// TIA Portal V20 export
DATA_BLOCK "HmiInterface"   // DB98
{ DB_Accessible_From_OPC_UA := 'FALSE' }
AUTHOR : ERsystem_FA2_DH. Kim
// stored: Access Published, DBAccessibleFromOPCUA false, DBAccessibleFromWebserver false, MemoryReserve 100, Namespace Unit1.Em5
   VAR
      em : "LAF_typeEmInterface";
      cm : Struct
         softCam : "Unit1.type_emRelations_em5_SoftCam";
         brakeTest : Struct
            cathodeMainPnP1AxisZ : "LER_typeBrakeTestEmInterface";
            cathodeMainPnP2AxisZ : "LER_typeBrakeTestEmInterface";
         END_STRUCT;
      END_STRUCT;
      mainPnP : Struct
         jobs { S7_SetPoint := 'True'} : "LAF_typeJobsInterface";
         sequence { S7_SetPoint := 'True'} : "LAF_typeSequenceInterface";
      END_STRUCT;
      alignTable : Struct
         jobs { S7_SetPoint := 'True'} : "LAF_typeJobsInterface";
         sequence { S7_SetPoint := 'True'} : "LAF_typeSequenceInterface";
      END_STRUCT;
      ngPnP : Struct
         jobs { S7_SetPoint := 'True'} : "LAF_typeJobsInterface";
         sequence { S7_SetPoint := 'True'} : "LAF_typeSequenceInterface";
      END_STRUCT;
      gaugeRnR : Struct
         jobs { S7_SetPoint := 'True'} : "LAF_typeJobsInterface";
         sequence { S7_SetPoint := 'True'} : "LAF_typeSequenceInterface";
      END_STRUCT;
      cathodeNgCount : "LER_typeAlarmCounterInterface";
      cmPnp1stCathodeDetect { S7_SetPoint := 'True'} : "LBC_typeDigitalSignalInterface";
      cmPnp2ndCathodeDetect { S7_SetPoint := 'True'} : "LBC_typeDigitalSignalInterface";
      cmCathodeAlignTableElectrodeDetect { S7_SetPoint := 'True'} : "LBC_typeDigitalSignalInterface";
      cmCathodeNgPnpElectrodeDetect { S7_SetPoint := 'True'} : "LBC_typeDigitalSignalInterface";
      cmCathodeNgBoxFullSensorDetect { S7_SetPoint := 'True'} : "LBC_typeDigitalSignalInterface";
      cmCathodeNgBoxDetect { S7_SetPoint := 'True'} : "LBC_typeDigitalSignalInterface";
   END_VAR
   VAR RETAIN
      cmCathodeMainPnP1AxisX : "LBC_typeAxis64PosInterface";
      cmCathodeMainPnP2AxisX : "LBC_typeAxis64PosInterface";
      cmCathodeMainPnP1AxisY : "LBC_typeAxis64PosInterface";
      cmCathodeMainPnP1AxisZ : "LBC_typeAxis64PosInterface";
      cmCathodeMainPnP2AxisZ : "LBC_typeAxis64PosInterface";
      cmCathodeAlignTableAxisX : "LBC_typeAxis64PosInterface";
      cmCathodeAlignTableAxisY1 : "LBC_typeAxis64PosInterface";
      cmCathodeAlignTableAxisY2 : "LBC_typeAxis64PosInterface";
   END_VAR
   VAR
      cmCathodeMainPnP1RotaryCwCcw : "LBC_typeTwoWayActuatorInterface";
      cmCathodeMainPnP1SuctionPlateVacuum : "LBC_typeTwoWayActuatorInterface";
      cmCathodeMainPnP2SuctionPlateVacuum : "LBC_typeTwoWayActuatorInterface";
      cmCathodeAlignTableSuctionPlateVacuum : "LBC_typeTwoWayActuatorInterface";
      cmCathodeGlassCleaning : "LBC_typeTwoWayActuatorInterface";
      cmCathodeNgPnpUpDown : "LBC_typeTwoWayActuatorInterface";
      cmCathodeNgPnp1stFwdBwd : "LBC_typeTwoWayActuatorInterface";
      cmCathodeNgPnp2ndFwdBwd { S7_SetPoint := 'True'} : "LBC_typeTwoWayActuatorInterface";
      cmCathodeMaintenanceMovingFixFrontRearFwdBwd : "LBC_typeTwoWayActuatorInterface";
      cmCathodeNgBoxLiftUpDown { S7_SetPoint := 'True'} : "LBC_typeTwoWayActuatorInterface";
      cmCathodeNgBoxLockUpDown { S7_SetPoint := 'True'} : "LBC_typeTwoWayActuatorInterface";
      cmCathodeNgPnpVaccum : "LBC_typeTwoWayActuatorInterface";
      cmCathodeConveyorCoverFwdBwd { S7_SetPoint := 'True'} : "LBC_typeTwoWayActuatorInterface";
      cmCathodeConveyorPickUpBlower { S7_SetPoint := 'True'} : "LBC_typeTwoWayActuatorInterface";
      cmAlignVisionControllerInterface : "LER_typeVisionInterface";
      AlignVisionHistory : "LER_typeVisionHistory";
      AlignVisionConversion : "LER_typeVisionAlignResultData";
      AlignCalibration : "LER_typeAlignCalibrationInterface";
      AlignMoveCalibration : "LER_typeAlignMoveCalibrationInterface";
      AlignThetaCalibration { S7_SetPoint := 'True'} : "LER_typeAlignThetaCalibrationInterface";
      AlignSyncMove : "LER_typeAlignSyncMoveInterface";
   END_VAR
   VAR RETAIN
      GaugeRnR1Align : "LER_typeCount";
   END_VAR
   VAR
      GaugeRnR1Stack { S7_SetPoint := 'True'} : "LER_typeCount";
      GaugeRnR3Align { S7_SetPoint := 'True'} : "LER_typeCount";
      intCondition : Struct
         Axis_07 { S7_SetPoint := 'True'} : "LER.typeAxisIntlockAll";   // CathodeMainPnP1AxisX
         Axis_08 { S7_SetPoint := 'True'} : "LER.typeAxisIntlockAll";   // CathodeMainPnP2AxisX
         Axis_09 { S7_SetPoint := 'True'} : "LER.typeAxisIntlockAll";   // CathodeMainPnP1AxisY
         Axis_10 { S7_SetPoint := 'True'} : "LER.typeAxisIntlockAll";   // CathodeMainPnP1AxisZ
         Axis_13 { S7_SetPoint := 'True'} : "LER.typeAxisIntlockAll";   // CathodeMainPnP2AxisZ
         Axis_18 { S7_SetPoint := 'True'} : "LER.typeAxisIntlockAll";   // CathodeAlignTableAxisX
         Axis_19 { S7_SetPoint := 'True'} : "LER.typeAxisIntlockAll";   // CathodeAlignTableAxisY1
         Axis_20 { S7_SetPoint := 'True'} : "LER.typeAxisIntlockAll";   // CathodeAlignTableAxisY2
         Actuator_23 : "LER.typeAxisActuatorCondition";   // CathodeMaintenanceMovingFixFrontFwdBwd
         Actuator_24 : "LER.typeAxisActuatorCondition";   // SP
         Actuator_25 : "LER.typeAxisActuatorCondition";   // CathodeNgBoxLockUpDown
         Actuator_26 : "LER.typeAxisActuatorCondition";   // CathodeNgBoxLiftUpDown
         Actuator_27 : "LER.typeAxisActuatorCondition";   // CathodeNgPnp2ndFwdBwd
         Actuator_28 : "LER.typeAxisActuatorCondition";   // SP
         Actuator_29 : "LER.typeAxisActuatorCondition";   // CathodeNgPnpUpDown
         Actuator_30 : "LER.typeAxisActuatorCondition";   // CathodeGlassCleaning
         Actuator_31 : "LER.typeAxisActuatorCondition";   // CathodeMainPnP1RotaryCwCcw
         Actuator_32 : "LER.typeAxisActuatorCondition";   // CathodeNgPnp1stFwdBwd
      END_STRUCT;
   END_VAR
BEGIN
   em.interlinkMode.link := FALSE;
   em.interlinkMode.unlink := FALSE;
   em.interlinkMode.isLinked := TRUE;
   em.commands.enable := FALSE;
   em.commands.acknowledge := FALSE;
   em.commands.disableAlarms := FALSE;
   em.commands.activateSimulation := FALSE;
   em.commands.home := FALSE;
   em.commands.moveToInitialPosition := FALSE;
   em.commands.directModeControl := 16#0000_0001;
   em.commands.directStateControl := 16#0000_0004;
   em.status.enabled := TRUE;
   em.status.acknowledgeActive := FALSE;
   em.status.alarmsDisabled := FALSE;
   em.status.simulationActive := TRUE;
   em.status.safetyReleased := TRUE;
   em.status.initialized := TRUE;
   em.status.homed := FALSE;
   em.status.safeState := FALSE;
   em.status.stateComplete := FALSE;
   em.alarms.error := FALSE;
   em.alarms.warning := TRUE;
   em.alarms.info := FALSE;
   em.alarms.home := FALSE;
   cm.softCam.cathodeMainPnP1AxisX.reelCutConveyerPos.inPos := FALSE;
   cm.softCam.cathodeMainPnP1AxisX.reelCutConveyerPos.isBefore := FALSE;
   cm.softCam.cathodeMainPnP1AxisX.reelCutConveyerPos.isAfter := TRUE;
   cm.softCam.cathodeMainPnP1AxisX.alignTablePos.inPos := TRUE;
   cm.softCam.cathodeMainPnP1AxisX.alignTablePos.isBefore := FALSE;
   cm.softCam.cathodeMainPnP1AxisX.alignTablePos.isAfter := FALSE;
   cm.softCam.cathodeMainPnP1AxisX.Pos2.inPos := FALSE;
   cm.softCam.cathodeMainPnP1AxisX.Pos2.isBefore := TRUE;
   cm.softCam.cathodeMainPnP1AxisX.Pos2.isAfter := FALSE;
   cm.softCam.cathodeMainPnP1AxisX.Pos3.inPos := FALSE;
   cm.softCam.cathodeMainPnP1AxisX.Pos3.isBefore := FALSE;
   cm.softCam.cathodeMainPnP1AxisX.Pos3.isAfter := TRUE;
   cm.softCam.cathodeMainPnP1AxisX.Pos4.inPos := FALSE;
   cm.softCam.cathodeMainPnP1AxisX.Pos4.isBefore := FALSE;
   cm.softCam.cathodeMainPnP1AxisX.Pos4.isAfter := TRUE;
   cm.softCam.cathodeMainPnP1AxisX.Pos5.inPos := FALSE;
   cm.softCam.cathodeMainPnP1AxisX.Pos5.isBefore := FALSE;
   cm.softCam.cathodeMainPnP1AxisX.Pos5.isAfter := TRUE;
   cm.softCam.cathodeMainPnP1AxisX.Pos6.inPos := FALSE;
   cm.softCam.cathodeMainPnP1AxisX.Pos6.isBefore := FALSE;
   cm.softCam.cathodeMainPnP1AxisX.Pos6.isAfter := TRUE;
   cm.softCam.cathodeMainPnP1AxisX.Pos7.inPos := FALSE;
   cm.softCam.cathodeMainPnP1AxisX.Pos7.isBefore := FALSE;
   cm.softCam.cathodeMainPnP1AxisX.Pos7.isAfter := TRUE;
   cm.softCam.cathodeMainPnP1AxisX.Pos8.inPos := FALSE;
   cm.softCam.cathodeMainPnP1AxisX.Pos8.isBefore := FALSE;
   cm.softCam.cathodeMainPnP1AxisX.Pos8.isAfter := TRUE;
   cm.softCam.cathodeMainPnP1AxisX.Pos9.inPos := FALSE;
   cm.softCam.cathodeMainPnP1AxisX.Pos9.isBefore := FALSE;
   cm.softCam.cathodeMainPnP1AxisX.Pos9.isAfter := TRUE;
   cm.softCam.cathodeMainPnP1AxisX.Pos10.inPos := FALSE;
   cm.softCam.cathodeMainPnP1AxisX.Pos10.isBefore := FALSE;
   cm.softCam.cathodeMainPnP1AxisX.Pos10.isAfter := TRUE;
   cm.softCam.cathodeMainPnP1AxisX.Pos11.inPos := FALSE;
   cm.softCam.cathodeMainPnP1AxisX.Pos11.isBefore := FALSE;
   cm.softCam.cathodeMainPnP1AxisX.Pos11.isAfter := TRUE;
   cm.softCam.cathodeMainPnP1AxisX.Pos12.inPos := FALSE;
   cm.softCam.cathodeMainPnP1AxisX.Pos12.isBefore := FALSE;
   cm.softCam.cathodeMainPnP1AxisX.Pos12.isAfter := TRUE;
   cm.softCam.cathodeMainPnP1AxisX.Pos13.inPos := FALSE;
   cm.softCam.cathodeMainPnP1AxisX.Pos13.isBefore := FALSE;
   cm.softCam.cathodeMainPnP1AxisX.Pos13.isAfter := TRUE;
   cm.softCam.cathodeMainPnP1AxisX.Pos14.inPos := FALSE;
   cm.softCam.cathodeMainPnP1AxisX.Pos14.isBefore := FALSE;
   cm.softCam.cathodeMainPnP1AxisX.Pos14.isAfter := TRUE;
   cm.softCam.cathodeMainPnP1AxisX.Pos15.inPos := FALSE;
   cm.softCam.cathodeMainPnP1AxisX.Pos15.isBefore := FALSE;
   cm.softCam.cathodeMainPnP1AxisX.Pos15.isAfter := TRUE;
   cm.softCam.cathodeMainPnP2AxisX.alignTablePos.inPos := FALSE;
   cm.softCam.cathodeMainPnP2AxisX.alignTablePos.isBefore := FALSE;
   cm.softCam.cathodeMainPnP2AxisX.alignTablePos.isAfter := TRUE;
   cm.softCam.cathodeMainPnP2AxisX.stackTablePos.inPos := TRUE;
   cm.softCam.cathodeMainPnP2AxisX.stackTablePos.isBefore := FALSE;
   cm.softCam.cathodeMainPnP2AxisX.stackTablePos.isAfter := FALSE;
   cm.softCam.cathodeMainPnP2AxisX.Pos2.inPos := FALSE;
   cm.softCam.cathodeMainPnP2AxisX.Pos2.isBefore := FALSE;
   cm.softCam.cathodeMainPnP2AxisX.Pos2.isAfter := TRUE;
   cm.softCam.cathodeMainPnP2AxisX.Pos3.inPos := FALSE;
   cm.softCam.cathodeMainPnP2AxisX.Pos3.isBefore := FALSE;
   cm.softCam.cathodeMainPnP2AxisX.Pos3.isAfter := TRUE;
   cm.softCam.cathodeMainPnP2AxisX.Pos4.inPos := FALSE;
   cm.softCam.cathodeMainPnP2AxisX.Pos4.isBefore := FALSE;
   cm.softCam.cathodeMainPnP2AxisX.Pos4.isAfter := TRUE;
   cm.softCam.cathodeMainPnP2AxisX.Pos5.inPos := FALSE;
   cm.softCam.cathodeMainPnP2AxisX.Pos5.isBefore := FALSE;
   cm.softCam.cathodeMainPnP2AxisX.Pos5.isAfter := TRUE;
   cm.softCam.cathodeMainPnP2AxisX.Pos6.inPos := FALSE;
   cm.softCam.cathodeMainPnP2AxisX.Pos6.isBefore := FALSE;
   cm.softCam.cathodeMainPnP2AxisX.Pos6.isAfter := TRUE;
   cm.softCam.cathodeMainPnP2AxisX.Pos7.inPos := FALSE;
   cm.softCam.cathodeMainPnP2AxisX.Pos7.isBefore := FALSE;
   cm.softCam.cathodeMainPnP2AxisX.Pos7.isAfter := TRUE;
   cm.softCam.cathodeMainPnP2AxisX.Pos8.inPos := FALSE;
   cm.softCam.cathodeMainPnP2AxisX.Pos8.isBefore := FALSE;
   cm.softCam.cathodeMainPnP2AxisX.Pos8.isAfter := TRUE;
   cm.softCam.cathodeMainPnP2AxisX.Pos9.inPos := FALSE;
   cm.softCam.cathodeMainPnP2AxisX.Pos9.isBefore := FALSE;
   cm.softCam.cathodeMainPnP2AxisX.Pos9.isAfter := TRUE;
   cm.softCam.cathodeMainPnP2AxisX.Pos10.inPos := FALSE;
   cm.softCam.cathodeMainPnP2AxisX.Pos10.isBefore := FALSE;
   cm.softCam.cathodeMainPnP2AxisX.Pos10.isAfter := TRUE;
   cm.softCam.cathodeMainPnP2AxisX.Pos11.inPos := FALSE;
   cm.softCam.cathodeMainPnP2AxisX.Pos11.isBefore := FALSE;
   cm.softCam.cathodeMainPnP2AxisX.Pos11.isAfter := TRUE;
   cm.softCam.cathodeMainPnP2AxisX.Pos12.inPos := FALSE;
   cm.softCam.cathodeMainPnP2AxisX.Pos12.isBefore := FALSE;
   cm.softCam.cathodeMainPnP2AxisX.Pos12.isAfter := TRUE;
   cm.softCam.cathodeMainPnP2AxisX.Pos13.inPos := FALSE;
   cm.softCam.cathodeMainPnP2AxisX.Pos13.isBefore := FALSE;
   cm.softCam.cathodeMainPnP2AxisX.Pos13.isAfter := TRUE;
   cm.softCam.cathodeMainPnP2AxisX.Pos14.inPos := FALSE;
   cm.softCam.cathodeMainPnP2AxisX.Pos14.isBefore := FALSE;
   cm.softCam.cathodeMainPnP2AxisX.Pos14.isAfter := TRUE;
   cm.softCam.cathodeMainPnP2AxisX.Pos15.inPos := FALSE;
   cm.softCam.cathodeMainPnP2AxisX.Pos15.isBefore := FALSE;
   cm.softCam.cathodeMainPnP2AxisX.Pos15.isAfter := TRUE;
   cm.softCam.cathodeMainPnP1AxisY.waitPos.inPos := TRUE;
   cm.softCam.cathodeMainPnP1AxisY.waitPos.isBefore := FALSE;
   cm.softCam.cathodeMainPnP1AxisY.waitPos.isAfter := FALSE;
   cm.softCam.cathodeMainPnP1AxisY.Pos1.inPos := TRUE;
   cm.softCam.cathodeMainPnP1AxisY.Pos1.isBefore := FALSE;
   cm.softCam.cathodeMainPnP1AxisY.Pos1.isAfter := FALSE;
   cm.softCam.cathodeMainPnP1AxisY.Pos2.inPos := TRUE;
   cm.softCam.cathodeMainPnP1AxisY.Pos2.isBefore := FALSE;
   cm.softCam.cathodeMainPnP1AxisY.Pos2.isAfter := FALSE;
   cm.softCam.cathodeMainPnP1AxisY.Pos3.inPos := TRUE;
   cm.softCam.cathodeMainPnP1AxisY.Pos3.isBefore := FALSE;
   cm.softCam.cathodeMainPnP1AxisY.Pos3.isAfter := FALSE;
   cm.softCam.cathodeMainPnP1AxisY.Pos4.inPos := TRUE;
   cm.softCam.cathodeMainPnP1AxisY.Pos4.isBefore := FALSE;
   cm.softCam.cathodeMainPnP1AxisY.Pos4.isAfter := FALSE;
   cm.softCam.cathodeMainPnP1AxisY.Pos5.inPos := TRUE;
   cm.softCam.cathodeMainPnP1AxisY.Pos5.isBefore := FALSE;
   cm.softCam.cathodeMainPnP1AxisY.Pos5.isAfter := FALSE;
   cm.softCam.cathodeMainPnP1AxisY.Pos6.inPos := TRUE;
   cm.softCam.cathodeMainPnP1AxisY.Pos6.isBefore := FALSE;
   cm.softCam.cathodeMainPnP1AxisY.Pos6.isAfter := FALSE;
   cm.softCam.cathodeMainPnP1AxisY.Pos7.inPos := TRUE;
   cm.softCam.cathodeMainPnP1AxisY.Pos7.isBefore := FALSE;
   cm.softCam.cathodeMainPnP1AxisY.Pos7.isAfter := FALSE;
   cm.softCam.cathodeMainPnP1AxisY.Pos8.inPos := TRUE;
   cm.softCam.cathodeMainPnP1AxisY.Pos8.isBefore := FALSE;
   cm.softCam.cathodeMainPnP1AxisY.Pos8.isAfter := FALSE;
   cm.softCam.cathodeMainPnP1AxisY.Pos9.inPos := TRUE;
   cm.softCam.cathodeMainPnP1AxisY.Pos9.isBefore := FALSE;
   cm.softCam.cathodeMainPnP1AxisY.Pos9.isAfter := FALSE;
   cm.softCam.cathodeMainPnP1AxisY.Pos10.inPos := TRUE;
   cm.softCam.cathodeMainPnP1AxisY.Pos10.isBefore := FALSE;
   cm.softCam.cathodeMainPnP1AxisY.Pos10.isAfter := FALSE;
   cm.softCam.cathodeMainPnP1AxisY.Pos11.inPos := TRUE;
   cm.softCam.cathodeMainPnP1AxisY.Pos11.isBefore := FALSE;
   cm.softCam.cathodeMainPnP1AxisY.Pos11.isAfter := FALSE;
   cm.softCam.cathodeMainPnP1AxisY.Pos12.inPos := TRUE;
   cm.softCam.cathodeMainPnP1AxisY.Pos12.isBefore := FALSE;
   cm.softCam.cathodeMainPnP1AxisY.Pos12.isAfter := FALSE;
   cm.softCam.cathodeMainPnP1AxisY.Pos13.inPos := TRUE;
   cm.softCam.cathodeMainPnP1AxisY.Pos13.isBefore := FALSE;
   cm.softCam.cathodeMainPnP1AxisY.Pos13.isAfter := FALSE;
   cm.softCam.cathodeMainPnP1AxisY.Pos14.inPos := TRUE;
   cm.softCam.cathodeMainPnP1AxisY.Pos14.isBefore := FALSE;
   cm.softCam.cathodeMainPnP1AxisY.Pos14.isAfter := FALSE;
   cm.softCam.cathodeMainPnP1AxisY.Pos15.inPos := TRUE;
   cm.softCam.cathodeMainPnP1AxisY.Pos15.isBefore := FALSE;
   cm.softCam.cathodeMainPnP1AxisY.Pos15.isAfter := FALSE;
   cm.softCam.cathodeMainPnP1AxisZ.upPos.inPos := FALSE;
   cm.softCam.cathodeMainPnP1AxisZ.upPos.isBefore := FALSE;
   cm.softCam.cathodeMainPnP1AxisZ.upPos.isAfter := TRUE;
   cm.softCam.cathodeMainPnP1AxisZ.reelCutConveyerDownPos.inPos := TRUE;
   cm.softCam.cathodeMainPnP1AxisZ.reelCutConveyerDownPos.isBefore := FALSE;
   cm.softCam.cathodeMainPnP1AxisZ.reelCutConveyerDownPos.isAfter := FALSE;
   cm.softCam.cathodeMainPnP1AxisZ.ailgnTableDownPos.inPos := TRUE;
   cm.softCam.cathodeMainPnP1AxisZ.ailgnTableDownPos.isBefore := FALSE;
   cm.softCam.cathodeMainPnP1AxisZ.ailgnTableDownPos.isAfter := FALSE;
   cm.softCam.cathodeMainPnP1AxisZ.avoidPos.inPos := FALSE;
   cm.softCam.cathodeMainPnP1AxisZ.avoidPos.isBefore := FALSE;
   cm.softCam.cathodeMainPnP1AxisZ.avoidPos.isAfter := TRUE;
   cm.softCam.cathodeMainPnP1AxisZ.Pos4.inPos := FALSE;
   cm.softCam.cathodeMainPnP1AxisZ.Pos4.isBefore := FALSE;
   cm.softCam.cathodeMainPnP1AxisZ.Pos4.isAfter := TRUE;
   cm.softCam.cathodeMainPnP1AxisZ.Pos5.inPos := FALSE;
   cm.softCam.cathodeMainPnP1AxisZ.Pos5.isBefore := FALSE;
   cm.softCam.cathodeMainPnP1AxisZ.Pos5.isAfter := TRUE;
   cm.softCam.cathodeMainPnP1AxisZ.Pos6.inPos := FALSE;
   cm.softCam.cathodeMainPnP1AxisZ.Pos6.isBefore := FALSE;
   cm.softCam.cathodeMainPnP1AxisZ.Pos6.isAfter := TRUE;
   cm.softCam.cathodeMainPnP1AxisZ.Pos7.inPos := FALSE;
   cm.softCam.cathodeMainPnP1AxisZ.Pos7.isBefore := FALSE;
   cm.softCam.cathodeMainPnP1AxisZ.Pos7.isAfter := TRUE;
   cm.softCam.cathodeMainPnP1AxisZ.Pos8.inPos := FALSE;
   cm.softCam.cathodeMainPnP1AxisZ.Pos8.isBefore := FALSE;
   cm.softCam.cathodeMainPnP1AxisZ.Pos8.isAfter := TRUE;
   cm.softCam.cathodeMainPnP1AxisZ.Pos9.inPos := FALSE;
   cm.softCam.cathodeMainPnP1AxisZ.Pos9.isBefore := FALSE;
   cm.softCam.cathodeMainPnP1AxisZ.Pos9.isAfter := TRUE;
   cm.softCam.cathodeMainPnP1AxisZ.Pos10.inPos := FALSE;
   cm.softCam.cathodeMainPnP1AxisZ.Pos10.isBefore := FALSE;
   cm.softCam.cathodeMainPnP1AxisZ.Pos10.isAfter := TRUE;
   cm.softCam.cathodeMainPnP1AxisZ.Pos11.inPos := FALSE;
   cm.softCam.cathodeMainPnP1AxisZ.Pos11.isBefore := FALSE;
   cm.softCam.cathodeMainPnP1AxisZ.Pos11.isAfter := TRUE;
   cm.softCam.cathodeMainPnP1AxisZ.Pos12.inPos := FALSE;
   cm.softCam.cathodeMainPnP1AxisZ.Pos12.isBefore := FALSE;
   cm.softCam.cathodeMainPnP1AxisZ.Pos12.isAfter := TRUE;
   cm.softCam.cathodeMainPnP1AxisZ.Pos13.inPos := FALSE;
   cm.softCam.cathodeMainPnP1AxisZ.Pos13.isBefore := FALSE;
   cm.softCam.cathodeMainPnP1AxisZ.Pos13.isAfter := TRUE;
   cm.softCam.cathodeMainPnP1AxisZ.Pos14.inPos := FALSE;
   cm.softCam.cathodeMainPnP1AxisZ.Pos14.isBefore := FALSE;
   cm.softCam.cathodeMainPnP1AxisZ.Pos14.isAfter := TRUE;
   cm.softCam.cathodeMainPnP1AxisZ.Pos15.inPos := FALSE;
   cm.softCam.cathodeMainPnP1AxisZ.Pos15.isBefore := FALSE;
   cm.softCam.cathodeMainPnP1AxisZ.Pos15.isAfter := TRUE;
   cm.softCam.cathodeMainPnP2AxisZ.upPos.inPos := FALSE;
   cm.softCam.cathodeMainPnP2AxisZ.upPos.isBefore := FALSE;
   cm.softCam.cathodeMainPnP2AxisZ.upPos.isAfter := TRUE;
   cm.softCam.cathodeMainPnP2AxisZ.ailgnTableDownPos.inPos := TRUE;
   cm.softCam.cathodeMainPnP2AxisZ.ailgnTableDownPos.isBefore := FALSE;
   cm.softCam.cathodeMainPnP2AxisZ.ailgnTableDownPos.isAfter := FALSE;
   cm.softCam.cathodeMainPnP2AxisZ.stackTableDownPos.inPos := TRUE;
   cm.softCam.cathodeMainPnP2AxisZ.stackTableDownPos.isBefore := FALSE;
   cm.softCam.cathodeMainPnP2AxisZ.stackTableDownPos.isAfter := FALSE;
   cm.softCam.cathodeMainPnP2AxisZ.avoidPos.inPos := FALSE;
   cm.softCam.cathodeMainPnP2AxisZ.avoidPos.isBefore := FALSE;
   cm.softCam.cathodeMainPnP2AxisZ.avoidPos.isAfter := TRUE;
   cm.softCam.cathodeMainPnP2AxisZ.Pos4.inPos := FALSE;
   cm.softCam.cathodeMainPnP2AxisZ.Pos4.isBefore := FALSE;
   cm.softCam.cathodeMainPnP2AxisZ.Pos4.isAfter := TRUE;
   cm.softCam.cathodeMainPnP2AxisZ.Pos5.inPos := FALSE;
   cm.softCam.cathodeMainPnP2AxisZ.Pos5.isBefore := FALSE;
   cm.softCam.cathodeMainPnP2AxisZ.Pos5.isAfter := TRUE;
   cm.softCam.cathodeMainPnP2AxisZ.Pos6.inPos := FALSE;
   cm.softCam.cathodeMainPnP2AxisZ.Pos6.isBefore := FALSE;
   cm.softCam.cathodeMainPnP2AxisZ.Pos6.isAfter := TRUE;
   cm.softCam.cathodeMainPnP2AxisZ.Pos7.inPos := FALSE;
   cm.softCam.cathodeMainPnP2AxisZ.Pos7.isBefore := FALSE;
   cm.softCam.cathodeMainPnP2AxisZ.Pos7.isAfter := TRUE;
   cm.softCam.cathodeMainPnP2AxisZ.Pos8.inPos := FALSE;
   cm.softCam.cathodeMainPnP2AxisZ.Pos8.isBefore := FALSE;
   cm.softCam.cathodeMainPnP2AxisZ.Pos8.isAfter := TRUE;
   cm.softCam.cathodeMainPnP2AxisZ.Pos9.inPos := FALSE;
   cm.softCam.cathodeMainPnP2AxisZ.Pos9.isBefore := FALSE;
   cm.softCam.cathodeMainPnP2AxisZ.Pos9.isAfter := TRUE;
   cm.softCam.cathodeMainPnP2AxisZ.Pos10.inPos := FALSE;
   cm.softCam.cathodeMainPnP2AxisZ.Pos10.isBefore := FALSE;
   cm.softCam.cathodeMainPnP2AxisZ.Pos10.isAfter := TRUE;
   cm.softCam.cathodeMainPnP2AxisZ.Pos11.inPos := FALSE;
   cm.softCam.cathodeMainPnP2AxisZ.Pos11.isBefore := FALSE;
   cm.softCam.cathodeMainPnP2AxisZ.Pos11.isAfter := TRUE;
   cm.softCam.cathodeMainPnP2AxisZ.Pos12.inPos := FALSE;
   cm.softCam.cathodeMainPnP2AxisZ.Pos12.isBefore := FALSE;
   cm.softCam.cathodeMainPnP2AxisZ.Pos12.isAfter := TRUE;
   cm.softCam.cathodeMainPnP2AxisZ.Pos13.inPos := FALSE;
   cm.softCam.cathodeMainPnP2AxisZ.Pos13.isBefore := FALSE;
   cm.softCam.cathodeMainPnP2AxisZ.Pos13.isAfter := TRUE;
   cm.softCam.cathodeMainPnP2AxisZ.Pos14.inPos := FALSE;
   cm.softCam.cathodeMainPnP2AxisZ.Pos14.isBefore := FALSE;
   cm.softCam.cathodeMainPnP2AxisZ.Pos14.isAfter := TRUE;
   cm.softCam.cathodeMainPnP2AxisZ.Pos15.inPos := FALSE;
   cm.softCam.cathodeMainPnP2AxisZ.Pos15.isBefore := FALSE;
   cm.softCam.cathodeMainPnP2AxisZ.Pos15.isAfter := TRUE;
   cm.softCam.cathodeAlignTableAxisX.waitPos.inPos := TRUE;
   cm.softCam.cathodeAlignTableAxisX.waitPos.isBefore := FALSE;
   cm.softCam.cathodeAlignTableAxisX.waitPos.isAfter := FALSE;
   cm.softCam.cathodeAlignTableAxisX.adjustPos.inPos := FALSE;
   cm.softCam.cathodeAlignTableAxisX.adjustPos.isBefore := TRUE;
   cm.softCam.cathodeAlignTableAxisX.adjustPos.isAfter := FALSE;
   cm.softCam.cathodeAlignTableAxisX.Pos2.inPos := FALSE;
   cm.softCam.cathodeAlignTableAxisX.Pos2.isBefore := TRUE;
   cm.softCam.cathodeAlignTableAxisX.Pos2.isAfter := FALSE;
   cm.softCam.cathodeAlignTableAxisX.Pos3.inPos := FALSE;
   cm.softCam.cathodeAlignTableAxisX.Pos3.isBefore := TRUE;
   cm.softCam.cathodeAlignTableAxisX.Pos3.isAfter := FALSE;
   cm.softCam.cathodeAlignTableAxisX.Pos4.inPos := FALSE;
   cm.softCam.cathodeAlignTableAxisX.Pos4.isBefore := FALSE;
   cm.softCam.cathodeAlignTableAxisX.Pos4.isAfter := TRUE;
   cm.softCam.cathodeAlignTableAxisX.Pos5.inPos := FALSE;
   cm.softCam.cathodeAlignTableAxisX.Pos5.isBefore := FALSE;
   cm.softCam.cathodeAlignTableAxisX.Pos5.isAfter := TRUE;
   cm.softCam.cathodeAlignTableAxisX.Pos6.inPos := FALSE;
   cm.softCam.cathodeAlignTableAxisX.Pos6.isBefore := FALSE;
   cm.softCam.cathodeAlignTableAxisX.Pos6.isAfter := TRUE;
   cm.softCam.cathodeAlignTableAxisX.Pos7.inPos := FALSE;
   cm.softCam.cathodeAlignTableAxisX.Pos7.isBefore := FALSE;
   cm.softCam.cathodeAlignTableAxisX.Pos7.isAfter := TRUE;
   cm.softCam.cathodeAlignTableAxisX.Pos8.inPos := FALSE;
   cm.softCam.cathodeAlignTableAxisX.Pos8.isBefore := FALSE;
   cm.softCam.cathodeAlignTableAxisX.Pos8.isAfter := TRUE;
   cm.softCam.cathodeAlignTableAxisX.Pos9.inPos := FALSE;
   cm.softCam.cathodeAlignTableAxisX.Pos9.isBefore := TRUE;
   cm.softCam.cathodeAlignTableAxisX.Pos9.isAfter := FALSE;
   cm.softCam.cathodeAlignTableAxisX.Pos10.inPos := TRUE;
   cm.softCam.cathodeAlignTableAxisX.Pos10.isBefore := FALSE;
   cm.softCam.cathodeAlignTableAxisX.Pos10.isAfter := FALSE;
   cm.softCam.cathodeAlignTableAxisX.Pos11.inPos := TRUE;
   cm.softCam.cathodeAlignTableAxisX.Pos11.isBefore := FALSE;
   cm.softCam.cathodeAlignTableAxisX.Pos11.isAfter := FALSE;
   cm.softCam.cathodeAlignTableAxisX.Pos12.inPos := TRUE;
   cm.softCam.cathodeAlignTableAxisX.Pos12.isBefore := FALSE;
   cm.softCam.cathodeAlignTableAxisX.Pos12.isAfter := FALSE;
   cm.softCam.cathodeAlignTableAxisX.Pos13.inPos := TRUE;
   cm.softCam.cathodeAlignTableAxisX.Pos13.isBefore := FALSE;
   cm.softCam.cathodeAlignTableAxisX.Pos13.isAfter := FALSE;
   cm.softCam.cathodeAlignTableAxisX.Pos14.inPos := TRUE;
   cm.softCam.cathodeAlignTableAxisX.Pos14.isBefore := FALSE;
   cm.softCam.cathodeAlignTableAxisX.Pos14.isAfter := FALSE;
   cm.softCam.cathodeAlignTableAxisX.Pos15.inPos := TRUE;
   cm.softCam.cathodeAlignTableAxisX.Pos15.isBefore := FALSE;
   cm.softCam.cathodeAlignTableAxisX.Pos15.isAfter := FALSE;
   cm.softCam.cathodeAlignTableAxisY1.waitPos.inPos := TRUE;
   cm.softCam.cathodeAlignTableAxisY1.waitPos.isBefore := FALSE;
   cm.softCam.cathodeAlignTableAxisY1.waitPos.isAfter := FALSE;
   cm.softCam.cathodeAlignTableAxisY1.adjustPos.inPos := FALSE;
   cm.softCam.cathodeAlignTableAxisY1.adjustPos.isBefore := TRUE;
   cm.softCam.cathodeAlignTableAxisY1.adjustPos.isAfter := FALSE;
   cm.softCam.cathodeAlignTableAxisY1.Pos2.inPos := FALSE;
   cm.softCam.cathodeAlignTableAxisY1.Pos2.isBefore := TRUE;
   cm.softCam.cathodeAlignTableAxisY1.Pos2.isAfter := FALSE;
   cm.softCam.cathodeAlignTableAxisY1.Pos3.inPos := FALSE;
   cm.softCam.cathodeAlignTableAxisY1.Pos3.isBefore := TRUE;
   cm.softCam.cathodeAlignTableAxisY1.Pos3.isAfter := FALSE;
   cm.softCam.cathodeAlignTableAxisY1.Pos4.inPos := FALSE;
   cm.softCam.cathodeAlignTableAxisY1.Pos4.isBefore := TRUE;
   cm.softCam.cathodeAlignTableAxisY1.Pos4.isAfter := FALSE;
   cm.softCam.cathodeAlignTableAxisY1.Pos5.inPos := FALSE;
   cm.softCam.cathodeAlignTableAxisY1.Pos5.isBefore := TRUE;
   cm.softCam.cathodeAlignTableAxisY1.Pos5.isAfter := FALSE;
   cm.softCam.cathodeAlignTableAxisY1.Pos6.inPos := FALSE;
   cm.softCam.cathodeAlignTableAxisY1.Pos6.isBefore := TRUE;
   cm.softCam.cathodeAlignTableAxisY1.Pos6.isAfter := FALSE;
   cm.softCam.cathodeAlignTableAxisY1.Pos7.inPos := FALSE;
   cm.softCam.cathodeAlignTableAxisY1.Pos7.isBefore := FALSE;
   cm.softCam.cathodeAlignTableAxisY1.Pos7.isAfter := TRUE;
   cm.softCam.cathodeAlignTableAxisY1.Pos8.inPos := FALSE;
   cm.softCam.cathodeAlignTableAxisY1.Pos8.isBefore := TRUE;
   cm.softCam.cathodeAlignTableAxisY1.Pos8.isAfter := FALSE;
   cm.softCam.cathodeAlignTableAxisY1.Pos9.inPos := FALSE;
   cm.softCam.cathodeAlignTableAxisY1.Pos9.isBefore := FALSE;
   cm.softCam.cathodeAlignTableAxisY1.Pos9.isAfter := TRUE;
   cm.softCam.cathodeAlignTableAxisY1.Pos10.inPos := TRUE;
   cm.softCam.cathodeAlignTableAxisY1.Pos10.isBefore := FALSE;
   cm.softCam.cathodeAlignTableAxisY1.Pos10.isAfter := FALSE;
   cm.softCam.cathodeAlignTableAxisY1.Pos11.inPos := TRUE;
   cm.softCam.cathodeAlignTableAxisY1.Pos11.isBefore := FALSE;
   cm.softCam.cathodeAlignTableAxisY1.Pos11.isAfter := FALSE;
   cm.softCam.cathodeAlignTableAxisY1.Pos12.inPos := TRUE;
   cm.softCam.cathodeAlignTableAxisY1.Pos12.isBefore := FALSE;
   cm.softCam.cathodeAlignTableAxisY1.Pos12.isAfter := FALSE;
   cm.softCam.cathodeAlignTableAxisY1.Pos13.inPos := TRUE;
   cm.softCam.cathodeAlignTableAxisY1.Pos13.isBefore := FALSE;
   cm.softCam.cathodeAlignTableAxisY1.Pos13.isAfter := FALSE;
   cm.softCam.cathodeAlignTableAxisY1.Pos14.inPos := TRUE;
   cm.softCam.cathodeAlignTableAxisY1.Pos14.isBefore := FALSE;
   cm.softCam.cathodeAlignTableAxisY1.Pos14.isAfter := FALSE;
   cm.softCam.cathodeAlignTableAxisY1.Pos15.inPos := TRUE;
   cm.softCam.cathodeAlignTableAxisY1.Pos15.isBefore := FALSE;
   cm.softCam.cathodeAlignTableAxisY1.Pos15.isAfter := FALSE;
   cm.softCam.cathodeAlignTableAxisY2.waitPos.inPos := TRUE;
   cm.softCam.cathodeAlignTableAxisY2.waitPos.isBefore := FALSE;
   cm.softCam.cathodeAlignTableAxisY2.waitPos.isAfter := FALSE;
   cm.softCam.cathodeAlignTableAxisY2.adjustPos.inPos := FALSE;
   cm.softCam.cathodeAlignTableAxisY2.adjustPos.isBefore := TRUE;
   cm.softCam.cathodeAlignTableAxisY2.adjustPos.isAfter := FALSE;
   cm.softCam.cathodeAlignTableAxisY2.Pos2.inPos := FALSE;
   cm.softCam.cathodeAlignTableAxisY2.Pos2.isBefore := FALSE;
   cm.softCam.cathodeAlignTableAxisY2.Pos2.isAfter := TRUE;
   cm.softCam.cathodeAlignTableAxisY2.Pos3.inPos := FALSE;
   cm.softCam.cathodeAlignTableAxisY2.Pos3.isBefore := FALSE;
   cm.softCam.cathodeAlignTableAxisY2.Pos3.isAfter := TRUE;
   cm.softCam.cathodeAlignTableAxisY2.Pos4.inPos := FALSE;
   cm.softCam.cathodeAlignTableAxisY2.Pos4.isBefore := FALSE;
   cm.softCam.cathodeAlignTableAxisY2.Pos4.isAfter := TRUE;
   cm.softCam.cathodeAlignTableAxisY2.Pos5.inPos := FALSE;
   cm.softCam.cathodeAlignTableAxisY2.Pos5.isBefore := FALSE;
   cm.softCam.cathodeAlignTableAxisY2.Pos5.isAfter := TRUE;
   cm.softCam.cathodeAlignTableAxisY2.Pos6.inPos := FALSE;
   cm.softCam.cathodeAlignTableAxisY2.Pos6.isBefore := FALSE;
   cm.softCam.cathodeAlignTableAxisY2.Pos6.isAfter := TRUE;
   cm.softCam.cathodeAlignTableAxisY2.Pos7.inPos := FALSE;
   cm.softCam.cathodeAlignTableAxisY2.Pos7.isBefore := TRUE;
   cm.softCam.cathodeAlignTableAxisY2.Pos7.isAfter := FALSE;
   cm.softCam.cathodeAlignTableAxisY2.Pos8.inPos := FALSE;
   cm.softCam.cathodeAlignTableAxisY2.Pos8.isBefore := FALSE;
   cm.softCam.cathodeAlignTableAxisY2.Pos8.isAfter := TRUE;
   cm.softCam.cathodeAlignTableAxisY2.Pos9.inPos := FALSE;
   cm.softCam.cathodeAlignTableAxisY2.Pos9.isBefore := TRUE;
   cm.softCam.cathodeAlignTableAxisY2.Pos9.isAfter := FALSE;
   cm.softCam.cathodeAlignTableAxisY2.Pos10.inPos := TRUE;
   cm.softCam.cathodeAlignTableAxisY2.Pos10.isBefore := FALSE;
   cm.softCam.cathodeAlignTableAxisY2.Pos10.isAfter := FALSE;
   cm.softCam.cathodeAlignTableAxisY2.Pos11.inPos := TRUE;
   cm.softCam.cathodeAlignTableAxisY2.Pos11.isBefore := FALSE;
   cm.softCam.cathodeAlignTableAxisY2.Pos11.isAfter := FALSE;
   cm.softCam.cathodeAlignTableAxisY2.Pos12.inPos := TRUE;
   cm.softCam.cathodeAlignTableAxisY2.Pos12.isBefore := FALSE;
   cm.softCam.cathodeAlignTableAxisY2.Pos12.isAfter := FALSE;
   cm.softCam.cathodeAlignTableAxisY2.Pos13.inPos := TRUE;
   cm.softCam.cathodeAlignTableAxisY2.Pos13.isBefore := FALSE;
   cm.softCam.cathodeAlignTableAxisY2.Pos13.isAfter := FALSE;
   cm.softCam.cathodeAlignTableAxisY2.Pos14.inPos := TRUE;
   cm.softCam.cathodeAlignTableAxisY2.Pos14.isBefore := FALSE;
   cm.softCam.cathodeAlignTableAxisY2.Pos14.isAfter := FALSE;
   cm.softCam.cathodeAlignTableAxisY2.Pos15.inPos := TRUE;
   cm.softCam.cathodeAlignTableAxisY2.Pos15.isBefore := FALSE;
   cm.softCam.cathodeAlignTableAxisY2.Pos15.isAfter := FALSE;
   cm.brakeTest.cathodeMainPnP1AxisZ.commands.start := FALSE;
   cm.brakeTest.cathodeMainPnP1AxisZ.commands.stop := FALSE;
   cm.brakeTest.cathodeMainPnP1AxisZ.monitoring.error := FALSE;
   cm.brakeTest.cathodeMainPnP1AxisZ.monitoring.ready := FALSE;
   cm.brakeTest.cathodeMainPnP1AxisZ.monitoring.busy := FALSE;
   cm.brakeTest.cathodeMainPnP1AxisZ.monitoring.complete := FALSE;
   cm.brakeTest.cathodeMainPnP1AxisZ.monitoring.brakeSelected := FALSE;
   cm.brakeTest.cathodeMainPnP1AxisZ.monitoring.brakeActive := FALSE;
   cm.brakeTest.cathodeMainPnP1AxisZ.monitoring.brakeResult := FALSE;
   cm.brakeTest.cathodeMainPnP1AxisZ.monitoring.brakeCompleted := FALSE;
   cm.brakeTest.cathodeMainPnP1AxisZ.monitoring."step" := 0;
   cm.brakeTest.cathodeMainPnP2AxisZ.commands.start := FALSE;
   cm.brakeTest.cathodeMainPnP2AxisZ.commands.stop := FALSE;
   cm.brakeTest.cathodeMainPnP2AxisZ.monitoring.error := FALSE;
   cm.brakeTest.cathodeMainPnP2AxisZ.monitoring.ready := FALSE;
   cm.brakeTest.cathodeMainPnP2AxisZ.monitoring.busy := FALSE;
   cm.brakeTest.cathodeMainPnP2AxisZ.monitoring.complete := FALSE;
   cm.brakeTest.cathodeMainPnP2AxisZ.monitoring.brakeSelected := FALSE;
   cm.brakeTest.cathodeMainPnP2AxisZ.monitoring.brakeActive := FALSE;
   cm.brakeTest.cathodeMainPnP2AxisZ.monitoring.brakeResult := FALSE;
   cm.brakeTest.cathodeMainPnP2AxisZ.monitoring.brakeCompleted := FALSE;
   cm.brakeTest.cathodeMainPnP2AxisZ.monitoring."step" := 0;
   mainPnP.jobs.commands.setJobNumber := 0;
   mainPnP.jobs.commands.reset := FALSE;
   mainPnP.jobs.status.activeJobNumber := 0;
   mainPnP.jobs.status.previousCycleJobNumber := 0;
   mainPnP.jobs.status.manualControlEnabled := FALSE;
   mainPnP.jobs.status.memoryJobTime := 16#0000_4E97_C5E2_6789;
   mainPnP.sequence.commands.setAutomaticMode := FALSE;
   mainPnP.sequence.commands.setSingleStepMode := FALSE;
   mainPnP.sequence.commands.off := FALSE;
   mainPnP.sequence.commands.initialize := FALSE;
   mainPnP.sequence.commands.start := FALSE;
   mainPnP.sequence.commands.immediateStop := FALSE;
   mainPnP.sequence.commands.hold := FALSE;
   mainPnP.sequence.commands.nextStep := FALSE;
   mainPnP.sequence.commands.interlockStepChange := FALSE;
   mainPnP.sequence.monitoring.automaticMode := TRUE;
   mainPnP.sequence.monitoring.singleStepMode := FALSE;
   mainPnP.sequence.monitoring.currentStep := 1;
   mainPnP.sequence.monitoring.nextStep := 1;
   mainPnP.sequence.monitoring.previousStep := 190;
   mainPnP.sequence.monitoring.currentStepSTRING := 'N/A';
   mainPnP.sequence.monitoring.nextStepSTRING := 'N/A';
   mainPnP.sequence.monitoring.previousStepSTRING := 'N/A';
   mainPnP.sequence.monitoring.inStepIdle := TRUE;
   mainPnP.sequence.monitoring.inStepStopped := FALSE;
   mainPnP.sequence.monitoring.seqActive := TRUE;
   mainPnP.sequence.monitoring.stepActive := TRUE;
   mainPnP.sequence.monitoring.stepComplete := FALSE;
   mainPnP.sequence.monitoring.executionEnabled := TRUE;
   mainPnP.sequence.monitoring.initRequired := FALSE;
   mainPnP.sequence.monitoring.stepChangeReleased := TRUE;
   mainPnP.sequence.monitoring.justSteppedPulse := FALSE;
   mainPnP.sequence.monitoring.manualControlEnabled := FALSE;
   mainPnP.sequence.monitoring.manualModeChangeEnabled := FALSE;
   mainPnP.sequence.monitoring.memoryStepTimer := 16#0000_4E97_C5E1_A849;
   alignTable.jobs.commands.setJobNumber := 0;
   alignTable.jobs.commands.reset := FALSE;
   alignTable.jobs.status.activeJobNumber := 0;
   alignTable.jobs.status.previousCycleJobNumber := 0;
   alignTable.jobs.status.manualControlEnabled := FALSE;
   alignTable.jobs.status.memoryJobTime := 16#0000_4E98_3CE8_BA85;
   alignTable.sequence.commands.setAutomaticMode := FALSE;
   alignTable.sequence.commands.setSingleStepMode := FALSE;
   alignTable.sequence.commands.off := FALSE;
   alignTable.sequence.commands.initialize := FALSE;
   alignTable.sequence.commands.start := FALSE;
   alignTable.sequence.commands.immediateStop := FALSE;
   alignTable.sequence.commands.hold := FALSE;
   alignTable.sequence.commands.nextStep := FALSE;
   alignTable.sequence.commands.interlockStepChange := FALSE;
   alignTable.sequence.monitoring.automaticMode := TRUE;
   alignTable.sequence.monitoring.singleStepMode := FALSE;
   alignTable.sequence.monitoring.currentStep := 1;
   alignTable.sequence.monitoring.nextStep := 1;
   alignTable.sequence.monitoring.previousStep := 190;
   alignTable.sequence.monitoring.currentStepSTRING := 'N/A';
   alignTable.sequence.monitoring.nextStepSTRING := 'N/A';
   alignTable.sequence.monitoring.previousStepSTRING := 'N/A';
   alignTable.sequence.monitoring.inStepIdle := TRUE;
   alignTable.sequence.monitoring.inStepStopped := FALSE;
   alignTable.sequence.monitoring.seqActive := TRUE;
   alignTable.sequence.monitoring.stepActive := TRUE;
   alignTable.sequence.monitoring.stepComplete := FALSE;
   alignTable.sequence.monitoring.executionEnabled := TRUE;
   alignTable.sequence.monitoring.initRequired := FALSE;
   alignTable.sequence.monitoring.stepChangeReleased := TRUE;
   alignTable.sequence.monitoring.justSteppedPulse := FALSE;
   alignTable.sequence.monitoring.manualControlEnabled := FALSE;
   alignTable.sequence.monitoring.manualModeChangeEnabled := FALSE;
   alignTable.sequence.monitoring.memoryStepTimer := 16#0000_4E98_3CE8_0545;
   ngPnP.jobs.commands.setJobNumber := 0;
   ngPnP.jobs.commands.reset := FALSE;
   ngPnP.jobs.status.activeJobNumber := 0;
   ngPnP.jobs.status.previousCycleJobNumber := 0;
   ngPnP.jobs.status.manualControlEnabled := FALSE;
   ngPnP.jobs.status.memoryJobTime := 16#0000_4E8D_4269_263D;
   ngPnP.sequence.commands.setAutomaticMode := FALSE;
   ngPnP.sequence.commands.setSingleStepMode := FALSE;
   ngPnP.sequence.commands.off := FALSE;
   ngPnP.sequence.commands.initialize := FALSE;
   ngPnP.sequence.commands.start := FALSE;
   ngPnP.sequence.commands.immediateStop := FALSE;
   ngPnP.sequence.commands.hold := FALSE;
   ngPnP.sequence.commands.nextStep := FALSE;
   ngPnP.sequence.commands.interlockStepChange := FALSE;
   ngPnP.sequence.monitoring.automaticMode := TRUE;
   ngPnP.sequence.monitoring.singleStepMode := FALSE;
   ngPnP.sequence.monitoring.currentStep := 1;
   ngPnP.sequence.monitoring.nextStep := 1;
   ngPnP.sequence.monitoring.previousStep := 190;
   ngPnP.sequence.monitoring.currentStepSTRING := 'N/A';
   ngPnP.sequence.monitoring.nextStepSTRING := 'N/A';
   ngPnP.sequence.monitoring.previousStepSTRING := 'N/A';
   ngPnP.sequence.monitoring.inStepIdle := TRUE;
   ngPnP.sequence.monitoring.inStepStopped := FALSE;
   ngPnP.sequence.monitoring.seqActive := TRUE;
   ngPnP.sequence.monitoring.stepActive := TRUE;
   ngPnP.sequence.monitoring.stepComplete := FALSE;
   ngPnP.sequence.monitoring.executionEnabled := TRUE;
   ngPnP.sequence.monitoring.initRequired := FALSE;
   ngPnP.sequence.monitoring.stepChangeReleased := TRUE;
   ngPnP.sequence.monitoring.justSteppedPulse := FALSE;
   ngPnP.sequence.monitoring.manualControlEnabled := FALSE;
   ngPnP.sequence.monitoring.manualModeChangeEnabled := FALSE;
   ngPnP.sequence.monitoring.memoryStepTimer := 16#0000_4E8D_4268_74DE;
   gaugeRnR.jobs.commands.setJobNumber := 0;
   gaugeRnR.jobs.commands.reset := FALSE;
   gaugeRnR.jobs.status.activeJobNumber := 0;
   gaugeRnR.jobs.status.previousCycleJobNumber := 0;
   gaugeRnR.jobs.status.manualControlEnabled := FALSE;
   gaugeRnR.jobs.status.memoryJobTime := 0.0;
   gaugeRnR.sequence.commands.setAutomaticMode := FALSE;
   gaugeRnR.sequence.commands.setSingleStepMode := FALSE;
   gaugeRnR.sequence.commands.off := FALSE;
   gaugeRnR.sequence.commands.initialize := FALSE;
   gaugeRnR.sequence.commands.start := FALSE;
   gaugeRnR.sequence.commands.immediateStop := FALSE;
   gaugeRnR.sequence.commands.hold := FALSE;
   gaugeRnR.sequence.commands.nextStep := FALSE;
   gaugeRnR.sequence.commands.interlockStepChange := FALSE;
   gaugeRnR.sequence.monitoring.automaticMode := FALSE;
   gaugeRnR.sequence.monitoring.singleStepMode := FALSE;
   gaugeRnR.sequence.monitoring.currentStep := 0;
   gaugeRnR.sequence.monitoring.nextStep := 0;
   gaugeRnR.sequence.monitoring.previousStep := 0;
   gaugeRnR.sequence.monitoring.currentStepSTRING := '';
   gaugeRnR.sequence.monitoring.nextStepSTRING := '';
   gaugeRnR.sequence.monitoring.previousStepSTRING := '';
   gaugeRnR.sequence.monitoring.inStepIdle := FALSE;
   gaugeRnR.sequence.monitoring.inStepStopped := FALSE;
   gaugeRnR.sequence.monitoring.seqActive := FALSE;
   gaugeRnR.sequence.monitoring.stepActive := FALSE;
   gaugeRnR.sequence.monitoring.stepComplete := FALSE;
   gaugeRnR.sequence.monitoring.executionEnabled := FALSE;
   gaugeRnR.sequence.monitoring.initRequired := FALSE;
   gaugeRnR.sequence.monitoring.stepChangeReleased := FALSE;
   gaugeRnR.sequence.monitoring.justSteppedPulse := FALSE;
   gaugeRnR.sequence.monitoring.manualControlEnabled := FALSE;
   gaugeRnR.sequence.monitoring.manualModeChangeEnabled := FALSE;
   gaugeRnR.sequence.monitoring.memoryStepTimer := 0.0;
   cathodeNgCount.referenceDesignator := WSTRING#'Em5 Cathode NG Count';
   cathodeNgCount.actualCount := 0;
   cathodeNgCount.countResetButton := FALSE;
   cathodeNgCount.alarmSaveButton := FALSE;
   cathodeNgCount.ProcessValue.warningCount := 0;
   cathodeNgCount.ProcessValue.faultCount := 0;
   cathodeNgCount.SetValue.warningCount := 0;
   cathodeNgCount.SetValue.faultCount := 0;
   cmPnp1stCathodeDetect.commands.refreshConfiguration := FALSE;
   cmPnp1stCathodeDetect.commands.editConfiguration := FALSE;
   cmPnp1stCathodeDetect.commands.saveConfiguration := FALSE;
   cmPnp1stCathodeDetect.commands.reset := FALSE;
   cmPnp1stCathodeDetect.monitoring.enable := TRUE;
   cmPnp1stCathodeDetect.monitoring.referenceDesignator := WSTRING#'DigitalSignal';
   cmPnp1stCathodeDetect.monitoring.simulation := FALSE;
   cmPnp1stCathodeDetect.monitoring.processValue := FALSE;
   cmPnp1stCathodeDetect.monitoring.error := FALSE;
   cmPnp1stCathodeDetect.monitoring.status := 16#0000;
   cmPnp1stCathodeDetect.configuration.referenceDesignator := WSTRING#'DigitalSignal';
   cmPnp1stCathodeDetect.configuration.onDelay := T#0MS;
   cmPnp1stCathodeDetect.configuration.offDelay := T#0MS;
   cmPnp1stCathodeDetect.configuration.default := FALSE;
   cmPnp1stCathodeDetect.configuration.invertProcessValue := FALSE;
   cmPnp1stCathodeDetect.configuration.disableAlarms := FALSE;
   cmPnp2ndCathodeDetect.commands.refreshConfiguration := FALSE;
   cmPnp2ndCathodeDetect.commands.editConfiguration := FALSE;
   cmPnp2ndCathodeDetect.commands.saveConfiguration := FALSE;
   cmPnp2ndCathodeDetect.commands.reset := FALSE;
   cmPnp2ndCathodeDetect.monitoring.enable := TRUE;
   cmPnp2ndCathodeDetect.monitoring.referenceDesignator := WSTRING#'DigitalSignal';
   cmPnp2ndCathodeDetect.monitoring.simulation := FALSE;
   cmPnp2ndCathodeDetect.monitoring.processValue := FALSE;
   cmPnp2ndCathodeDetect.monitoring.error := FALSE;
   cmPnp2ndCathodeDetect.monitoring.status := 16#0000;
   cmPnp2ndCathodeDetect.configuration.referenceDesignator := WSTRING#'DigitalSignal';
   cmPnp2ndCathodeDetect.configuration.onDelay := T#0MS;
   cmPnp2ndCathodeDetect.configuration.offDelay := T#0MS;
   cmPnp2ndCathodeDetect.configuration.default := FALSE;
   cmPnp2ndCathodeDetect.configuration.invertProcessValue := FALSE;
   cmPnp2ndCathodeDetect.configuration.disableAlarms := FALSE;
   cmCathodeAlignTableElectrodeDetect.commands.refreshConfiguration := FALSE;
   cmCathodeAlignTableElectrodeDetect.commands.editConfiguration := FALSE;
   cmCathodeAlignTableElectrodeDetect.commands.saveConfiguration := FALSE;
   cmCathodeAlignTableElectrodeDetect.commands.reset := FALSE;
   cmCathodeAlignTableElectrodeDetect.monitoring.enable := TRUE;
   cmCathodeAlignTableElectrodeDetect.monitoring.referenceDesignator := WSTRING#'DigitalSignal';
   cmCathodeAlignTableElectrodeDetect.monitoring.simulation := FALSE;
   cmCathodeAlignTableElectrodeDetect.monitoring.processValue := FALSE;
   cmCathodeAlignTableElectrodeDetect.monitoring.error := FALSE;
   cmCathodeAlignTableElectrodeDetect.monitoring.status := 16#0000;
   cmCathodeAlignTableElectrodeDetect.configuration.referenceDesignator := WSTRING#'DigitalSignal';
   cmCathodeAlignTableElectrodeDetect.configuration.onDelay := T#0MS;
   cmCathodeAlignTableElectrodeDetect.configuration.offDelay := T#0MS;
   cmCathodeAlignTableElectrodeDetect.configuration.default := FALSE;
   cmCathodeAlignTableElectrodeDetect.configuration.invertProcessValue := FALSE;
   cmCathodeAlignTableElectrodeDetect.configuration.disableAlarms := FALSE;
   cmCathodeNgPnpElectrodeDetect.commands.refreshConfiguration := FALSE;
   cmCathodeNgPnpElectrodeDetect.commands.editConfiguration := FALSE;
   cmCathodeNgPnpElectrodeDetect.commands.saveConfiguration := FALSE;
   cmCathodeNgPnpElectrodeDetect.commands.reset := FALSE;
   cmCathodeNgPnpElectrodeDetect.monitoring.enable := FALSE;
   cmCathodeNgPnpElectrodeDetect.monitoring.referenceDesignator := WSTRING#'';
   cmCathodeNgPnpElectrodeDetect.monitoring.simulation := FALSE;
   cmCathodeNgPnpElectrodeDetect.monitoring.processValue := FALSE;
   cmCathodeNgPnpElectrodeDetect.monitoring.error := FALSE;
   cmCathodeNgPnpElectrodeDetect.monitoring.status := 16#0000;
   cmCathodeNgPnpElectrodeDetect.configuration.referenceDesignator := WSTRING#'DigitalSignal';
   cmCathodeNgPnpElectrodeDetect.configuration.onDelay := T#0MS;
   cmCathodeNgPnpElectrodeDetect.configuration.offDelay := T#0MS;
   cmCathodeNgPnpElectrodeDetect.configuration.default := FALSE;
   cmCathodeNgPnpElectrodeDetect.configuration.invertProcessValue := FALSE;
   cmCathodeNgPnpElectrodeDetect.configuration.disableAlarms := FALSE;
   cmCathodeNgBoxFullSensorDetect.commands.refreshConfiguration := FALSE;
   cmCathodeNgBoxFullSensorDetect.commands.editConfiguration := FALSE;
   cmCathodeNgBoxFullSensorDetect.commands.saveConfiguration := FALSE;
   cmCathodeNgBoxFullSensorDetect.commands.reset := FALSE;
   cmCathodeNgBoxFullSensorDetect.monitoring.enable := TRUE;
   cmCathodeNgBoxFullSensorDetect.monitoring.referenceDesignator := WSTRING#'DigitalSignal';
   cmCathodeNgBoxFullSensorDetect.monitoring.simulation := FALSE;
   cmCathodeNgBoxFullSensorDetect.monitoring.processValue := FALSE;
   cmCathodeNgBoxFullSensorDetect.monitoring.error := FALSE;
   cmCathodeNgBoxFullSensorDetect.monitoring.status := 16#0000;
   cmCathodeNgBoxFullSensorDetect.configuration.referenceDesignator := WSTRING#'DigitalSignal';
   cmCathodeNgBoxFullSensorDetect.configuration.onDelay := T#0MS;
   cmCathodeNgBoxFullSensorDetect.configuration.offDelay := T#0MS;
   cmCathodeNgBoxFullSensorDetect.configuration.default := FALSE;
   cmCathodeNgBoxFullSensorDetect.configuration.invertProcessValue := FALSE;
   cmCathodeNgBoxFullSensorDetect.configuration.disableAlarms := FALSE;
   cmCathodeNgBoxDetect.commands.refreshConfiguration := FALSE;
   cmCathodeNgBoxDetect.commands.editConfiguration := FALSE;
   cmCathodeNgBoxDetect.commands.saveConfiguration := FALSE;
   cmCathodeNgBoxDetect.commands.reset := FALSE;
   cmCathodeNgBoxDetect.monitoring.enable := TRUE;
   cmCathodeNgBoxDetect.monitoring.referenceDesignator := WSTRING#'DigitalSignal';
   cmCathodeNgBoxDetect.monitoring.simulation := FALSE;
   cmCathodeNgBoxDetect.monitoring.processValue := FALSE;
   cmCathodeNgBoxDetect.monitoring.error := FALSE;
   cmCathodeNgBoxDetect.monitoring.status := 16#0000;
   cmCathodeNgBoxDetect.configuration.referenceDesignator := WSTRING#'DigitalSignal';
   cmCathodeNgBoxDetect.configuration.onDelay := T#0MS;
   cmCathodeNgBoxDetect.configuration.offDelay := T#0MS;
   cmCathodeNgBoxDetect.configuration.default := FALSE;
   cmCathodeNgBoxDetect.configuration.invertProcessValue := FALSE;
   cmCathodeNgBoxDetect.configuration.disableAlarms := FALSE;
   cmCathodeMainPnP1AxisX.commandConfiguration.generalSettings.stopOnError := TRUE;
   cmCathodeMainPnP1AxisX.commandConfiguration.generalSettings.resetWithRestart := FALSE;
   cmCathodeMainPnP1AxisX.commandConfiguration.generalSettings.abortWaitingSyncCmd := TRUE;
   cmCathodeMainPnP1AxisX.commandConfiguration.power.startMode := 1;
   cmCathodeMainPnP1AxisX.commandConfiguration.power.stopMode := 0;
   cmCathodeMainPnP1AxisX.commandConfiguration.power.syncMotionSimulation := FALSE;
   cmCathodeMainPnP1AxisX.commandConfiguration.power.syncMotionSimulationExtendedMode := -1;
   cmCathodeMainPnP1AxisX.commandConfiguration.jog.velocity := 10.0;
   cmCathodeMainPnP1AxisX.commandConfiguration.jog.acceleration := 100.0;
   cmCathodeMainPnP1AxisX.commandConfiguration.jog.deceleration := 100.0;
   cmCathodeMainPnP1AxisX.commandConfiguration.jog.jerk := -1.0;
   cmCathodeMainPnP1AxisX.commandConfiguration.jog.positionControlled := TRUE;
   cmCathodeMainPnP1AxisX.commandConfiguration.jog.increment := 0.0;
   cmCathodeMainPnP1AxisX.commandConfiguration.jog.mode := 0;
   cmCathodeMainPnP1AxisX.commandConfiguration.moveVelocity.velocity := 10.0;
   cmCathodeMainPnP1AxisX.commandConfiguration.moveVelocity.acceleration := 100.0;
   cmCathodeMainPnP1AxisX.commandConfiguration.moveVelocity.deceleration := 100.0;
   cmCathodeMainPnP1AxisX.commandConfiguration.moveVelocity.jerk := -1.0;
   cmCathodeMainPnP1AxisX.commandConfiguration.moveVelocity.direction := 0;
   cmCathodeMainPnP1AxisX.commandConfiguration.moveVelocity.positionControlled := TRUE;
   cmCathodeMainPnP1AxisX.commandConfiguration.moveVelocity.velocityChangeOnTheFly := FALSE;
   cmCathodeMainPnP1AxisX.commandConfiguration.stop.deceleration := -1.0;
   cmCathodeMainPnP1AxisX.commandConfiguration.stop.jerk := -1.0;
   cmCathodeMainPnP1AxisX.commandConfiguration.stop.abortAcceleration := FALSE;
   cmCathodeMainPnP1AxisX.commandConfiguration.fastStop.deceleration := -1.0;
   cmCathodeMainPnP1AxisX.commandConfiguration.fastStop.jerk := -1.0;
   cmCathodeMainPnP1AxisX.commandConfiguration.fastStop.abortAcceleration := FALSE;
   cmCathodeMainPnP1AxisX.commandConfiguration.fastStop.replaceStopPossible := FALSE;
   cmCathodeMainPnP1AxisX.commandConfiguration.torqueLimiting.limit := -1.0;
   cmCathodeMainPnP1AxisX.commandConfiguration.torqueLimiting.mode := 0;
   cmCathodeMainPnP1AxisX.commandConfiguration.homing.position := 0.0;
   cmCathodeMainPnP1AxisX.commandConfiguration.homing.mode := 0;
   cmCathodeMainPnP1AxisX.commandConfiguration.homing.sensor := 0;
   cmCathodeMainPnP1AxisX.commandConfiguration.homing.extendedMode := -1;
   cmCathodeMainPnP1AxisX.commandConfiguration.homing.extendedModeTorqueLimit := 0.0;
   cmCathodeMainPnP1AxisX.commandConfiguration.homing.extendedModeTargetPosition := 0.0;
   cmCathodeMainPnP1AxisX.commandConfiguration.posRelative.distance := 0.0;
   cmCathodeMainPnP1AxisX.commandConfiguration.posRelative.velocity := 10.0;
   cmCathodeMainPnP1AxisX.commandConfiguration.posRelative.acceleration := 100.0;
   cmCathodeMainPnP1AxisX.commandConfiguration.posRelative.deceleration := 100.0;
   cmCathodeMainPnP1AxisX.commandConfiguration.posRelative.jerk := -1.0;
   cmCathodeMainPnP1AxisX.commandConfiguration.posRelative.direction := 0;
   cmCathodeMainPnP1AxisX.commandConfiguration.posAbsolute.position := 0.0;
   cmCathodeMainPnP1AxisX.commandConfiguration.posAbsolute.velocity := -1.0;
   cmCathodeMainPnP1AxisX.commandConfiguration.posAbsolute.acceleration := -1.0;
   cmCathodeMainPnP1AxisX.commandConfiguration.posAbsolute.deceleration := -1.0;
   cmCathodeMainPnP1AxisX.commandConfiguration.posAbsolute.jerk := 1382.07275733567;
   cmCathodeMainPnP1AxisX.commandConfiguration.posAbsolute.direction := 1;
   cmCathodeMainPnP1AxisX.commandConfiguration.posAbsolute.positionChangeOnTheFly := FALSE;
   cmCathodeMainPnP1AxisX.commandConfiguration.posAbsolute.velocityChangeOnTheFly := FALSE;
   cmCathodeMainPnP1AxisX.commandConfiguration.posSuperimposed.distance := 0.0;
   cmCathodeMainPnP1AxisX.commandConfiguration.posSuperimposed.velocityDiff := -1.0;
   cmCathodeMainPnP1AxisX.commandConfiguration.posSuperimposed.acceleration := -1.0;
   cmCathodeMainPnP1AxisX.commandConfiguration.posSuperimposed.deceleration := -1.0;
   cmCathodeMainPnP1AxisX.commandConfiguration.posSuperimposed.jerk := -1.0;
   cmCathodeMainPnP1AxisX.commandConfiguration.posSuperimposed.direction := 0;
   cmCathodeMainPnP1AxisX.commandConfiguration.haltSuperimposed.deceleration := -1.0;
   cmCathodeMainPnP1AxisX.commandConfiguration.haltSuperimposed.jerk := -1.0;
   cmCathodeMainPnP1AxisX.commandConfiguration.haltSuperimposed.abortAcceleration := FALSE;
   cmCathodeMainPnP1AxisX.commandConfiguration.gearInRelative.ratioNumerator := 1;
   cmCathodeMainPnP1AxisX.commandConfiguration.gearInRelative.ratioDenominator := 1;
   cmCathodeMainPnP1AxisX.commandConfiguration.gearInRelative.acceleration := -1.0;
   cmCathodeMainPnP1AxisX.commandConfiguration.gearInRelative.deceleration := -1.0;
   cmCathodeMainPnP1AxisX.commandConfiguration.gearInRelative.jerk := -1.0;
   cmCathodeMainPnP1AxisX.commandConfiguration.gearInRelative.ratioChangeOnTheFly := FALSE;
   cmCathodeMainPnP1AxisX.commandConfiguration.gearInAbsolute.ratioNumerator := 1;
   cmCathodeMainPnP1AxisX.commandConfiguration.gearInAbsolute.ratioDenominator := 1;
   cmCathodeMainPnP1AxisX.commandConfiguration.gearInAbsolute.masterSyncPosition := 0.0;
   cmCathodeMainPnP1AxisX.commandConfiguration.gearInAbsolute.slaveSyncPosition := 0.0;
   cmCathodeMainPnP1AxisX.commandConfiguration.gearInAbsolute.syncProfileReference := 1;
   cmCathodeMainPnP1AxisX.commandConfiguration.gearInAbsolute.masterStartDistance := 0.0;
   cmCathodeMainPnP1AxisX.commandConfiguration.gearInAbsolute.velocity := -1.0;
   cmCathodeMainPnP1AxisX.commandConfiguration.gearInAbsolute.acceleration := -1.0;
   cmCathodeMainPnP1AxisX.commandConfiguration.gearInAbsolute.deceleration := -1.0;
   cmCathodeMainPnP1AxisX.commandConfiguration.gearInAbsolute.jerk := -1.0;
   cmCathodeMainPnP1AxisX.commandConfiguration.gearInAbsolute.syncDirection := 1;
   cmCathodeMainPnP1AxisX.commandConfiguration.gearInAbsolute.ratioChangeOnTheFly := FALSE;
   cmCathodeMainPnP1AxisX.commandConfiguration.gearInVelocity.continuousUpdate := FALSE;
   cmCathodeMainPnP1AxisX.commandConfiguration.gearInVelocity.ratioNumerator := 1;
   cmCathodeMainPnP1AxisX.commandConfiguration.gearInVelocity.ratioDenominator := 1;
   cmCathodeMainPnP1AxisX.commandConfiguration.gearInVelocity.acceleration := -1.0;
   cmCathodeMainPnP1AxisX.commandConfiguration.gearInVelocity.deceleration := -1.0;
   cmCathodeMainPnP1AxisX.commandConfiguration.gearInVelocity.jerk := -1.0;
   cmCathodeMainPnP1AxisX.commandConfiguration.gearInVelocity.positionControlled := FALSE;
   cmCathodeMainPnP1AxisX.commandConfiguration.camIn.masterOffset := 0.0;
   cmCathodeMainPnP1AxisX.commandConfiguration.camIn.slaveOffset := 0.0;
   cmCathodeMainPnP1AxisX.commandConfiguration.camIn.masterScaling := 1.0;
   cmCathodeMainPnP1AxisX.commandConfiguration.camIn.slaveScaling := 1.0;
   cmCathodeMainPnP1AxisX.commandConfiguration.camIn.masterSyncPosition := 0.0;
   cmCathodeMainPnP1AxisX.commandConfiguration.camIn.syncProfileReference := 1;
   cmCathodeMainPnP1AxisX.commandConfiguration.camIn.masterStartDistance := 0.0;
   cmCathodeMainPnP1AxisX.commandConfiguration.camIn.velocity := -1.0;
   cmCathodeMainPnP1AxisX.commandConfiguration.camIn.acceleration := -1.0;
   cmCathodeMainPnP1AxisX.commandConfiguration.camIn.deceleration := -1.0;
   cmCathodeMainPnP1AxisX.commandConfiguration.camIn.jerk := -1.0;
   cmCathodeMainPnP1AxisX.commandConfiguration.camIn.applicationMode := 0;
   cmCathodeMainPnP1AxisX.commandConfiguration.camIn.syncDirection := 1;
   cmCathodeMainPnP1AxisX.commandConfiguration.gearOutCamOut.slavePosition := 0.0;
   cmCathodeMainPnP1AxisX.commandConfiguration.gearOutCamOut.syncProfileReference := 1;
   cmCathodeMainPnP1AxisX.commandConfiguration.gearOutCamOut.masterStopDistance := 0.0;
   cmCathodeMainPnP1AxisX.commandConfiguration.gearOutCamOut.deceleration := -1.0;
   cmCathodeMainPnP1AxisX.commandConfiguration.gearOutCamOut.jerk := -1.0;
   cmCathodeMainPnP1AxisX.commandConfiguration.gearOutCamOut.syncOutDirection := 3;
   cmCathodeMainPnP1AxisX.commandConfiguration.gearOutCamOut.gearOutCamOutMode := -1;
   cmCathodeMainPnP1AxisX.commandConfiguration.phasing.phaseShift := 0.0;
   cmCathodeMainPnP1AxisX.commandConfiguration.phasing.velocity := -1.0;
   cmCathodeMainPnP1AxisX.commandConfiguration.phasing.acceleration := -1.0;
   cmCathodeMainPnP1AxisX.commandConfiguration.phasing.deceleration := -1.0;
   cmCathodeMainPnP1AxisX.commandConfiguration.phasing.jerk := -1.0;
   cmCathodeMainPnP1AxisX.commandConfiguration.phasing.profileReference := 0;
   cmCathodeMainPnP1AxisX.commandConfiguration.phasing.phasingDistance := 0.0;
   cmCathodeMainPnP1AxisX.commandConfiguration.phasing.startPosition := 0.0;
   cmCathodeMainPnP1AxisX.commandConfiguration.phasing.direction := 3;
   cmCathodeMainPnP1AxisX.commandConfiguration.phasing.phaseAbsolute := TRUE;
   cmCathodeMainPnP1AxisX.commandConfiguration.phasing.phaseShiftChangeOnTheFly := FALSE;
   cmCathodeMainPnP1AxisX.commandConfiguration.offset.offset := 0.0;
   cmCathodeMainPnP1AxisX.commandConfiguration.offset.profileReference := 1;
   cmCathodeMainPnP1AxisX.commandConfiguration.offset.offsetDistance := 0.0;
   cmCathodeMainPnP1AxisX.commandConfiguration.offset.startPosition := 0.0;
   cmCathodeMainPnP1AxisX.commandConfiguration.offset.direction := 3;
   cmCathodeMainPnP1AxisX.commandConfiguration.offset.offsetAbsolute := TRUE;
   cmCathodeMainPnP1AxisX.commandConfiguration.offset.offsetChangeOnTheFly := FALSE;
   cmCathodeMainPnP1AxisX.commands.enableMasterControl := TRUE;
   cmCathodeMainPnP1AxisX.commands.enableAxis := FALSE;
   cmCathodeMainPnP1AxisX.commands.resetAxis := FALSE;
   cmCathodeMainPnP1AxisX.commands.openBrake := FALSE;
   cmCathodeMainPnP1AxisX.commands.jogForward := FALSE;
   cmCathodeMainPnP1AxisX.commands.jogBackward := FALSE;
   cmCathodeMainPnP1AxisX.commands.moveVelocity := FALSE;
   cmCathodeMainPnP1AxisX.commands.stop := FALSE;
   cmCathodeMainPnP1AxisX.commands.fastStop := FALSE;
   cmCathodeMainPnP1AxisX.commands.torqueLimiting := FALSE;
   cmCathodeMainPnP1AxisX.commands.homing := FALSE;
   cmCathodeMainPnP1AxisX.commands.posRelative := FALSE;
   cmCathodeMainPnP1AxisX.commands.posAbsolute := FALSE;
   cmCathodeMainPnP1AxisX.commands.posSuperimposed := FALSE;
   cmCathodeMainPnP1AxisX.commands.haltSuperimposed := FALSE;
   cmCathodeMainPnP1AxisX.commands.selectSetPosition := 0;
   cmCathodeMainPnP1AxisX.commands.uploadParameters := FALSE;
   cmCathodeMainPnP1AxisX.commands.refreshConfiguration := FALSE;
   cmCathodeMainPnP1AxisX.commands.editConfiguration := FALSE;
   cmCathodeMainPnP1AxisX.commands.saveConfiguration := FALSE;
   cmCathodeMainPnP1AxisX.commands.uploadCurrentTorque := FALSE;
   cmCathodeMainPnP1AxisX.commands.reset := FALSE;
   cmCathodeMainPnP1AxisX.monitoring.enable := TRUE;
   cmCathodeMainPnP1AxisX.monitoring.referenceDesignator := WSTRING#'CathodeMainPnP1AxisX';
   cmCathodeMainPnP1AxisX.monitoring.enabled := TRUE;
   cmCathodeMainPnP1AxisX.monitoring.enableManualCmds := FALSE;
   cmCathodeMainPnP1AxisX.monitoring.reset := FALSE;
   cmCathodeMainPnP1AxisX.monitoring.resetAxis := FALSE;
   cmCathodeMainPnP1AxisX.monitoring.enableAxis := TRUE;
   cmCathodeMainPnP1AxisX.monitoring.openBrake := FALSE;
   cmCathodeMainPnP1AxisX.monitoring.jogBackward := FALSE;
   cmCathodeMainPnP1AxisX.monitoring.jogForward := FALSE;
   cmCathodeMainPnP1AxisX.monitoring.moveVelocity := FALSE;
   cmCathodeMainPnP1AxisX.monitoring.stop := FALSE;
   cmCathodeMainPnP1AxisX.monitoring.fastStop := FALSE;
   cmCathodeMainPnP1AxisX.monitoring.torqueLimiting := FALSE;
   cmCathodeMainPnP1AxisX.monitoring.homing := FALSE;
   cmCathodeMainPnP1AxisX.monitoring.posRelative := FALSE;
   cmCathodeMainPnP1AxisX.monitoring.posAbsolute := FALSE;
   cmCathodeMainPnP1AxisX.monitoring.posSuperimposed := FALSE;
   cmCathodeMainPnP1AxisX.monitoring.haltSuperimposed := FALSE;
   cmCathodeMainPnP1AxisX.monitoring.brakeOpened := FALSE;
   cmCathodeMainPnP1AxisX.monitoring.axisEnabled := TRUE;
   cmCathodeMainPnP1AxisX.monitoring.resetActive := FALSE;
   cmCathodeMainPnP1AxisX.monitoring.inVelocity := FALSE;
   cmCathodeMainPnP1AxisX.monitoring.inLimitation := FALSE;
   cmCathodeMainPnP1AxisX.monitoring.inClamping := FALSE;
   cmCathodeMainPnP1AxisX.monitoring.startSync := FALSE;
   cmCathodeMainPnP1AxisX.monitoring.inSync := FALSE;
   cmCathodeMainPnP1AxisX.monitoring.inSimulation := FALSE;
   cmCathodeMainPnP1AxisX.monitoring.jogSelected := FALSE;
   cmCathodeMainPnP1AxisX.monitoring.moveVelocitySelected := FALSE;
   cmCathodeMainPnP1AxisX.monitoring.stopSelected := FALSE;
   cmCathodeMainPnP1AxisX.monitoring.fastStopSelected := FALSE;
   cmCathodeMainPnP1AxisX.monitoring.torqueLimitingSelected := FALSE;
   cmCathodeMainPnP1AxisX.monitoring.homingSelected := FALSE;
   cmCathodeMainPnP1AxisX.monitoring.posRelativeSelected := FALSE;
   cmCathodeMainPnP1AxisX.monitoring.posAbsoluteSelected := FALSE;
   cmCathodeMainPnP1AxisX.monitoring.posSuperimposedSelected := FALSE;
   cmCathodeMainPnP1AxisX.monitoring.haltSuperimposedSelected := FALSE;
   cmCathodeMainPnP1AxisX.monitoring.commandBusy := FALSE;
   cmCathodeMainPnP1AxisX.monitoring.commandDone := FALSE;
   cmCathodeMainPnP1AxisX.monitoring.commandAborted := FALSE;
   cmCathodeMainPnP1AxisX.monitoring.homingCommandBusy := FALSE;
   cmCathodeMainPnP1AxisX.monitoring.homingCommandDone := FALSE;
   cmCathodeMainPnP1AxisX.monitoring.homingCommandAborted := FALSE;
   cmCathodeMainPnP1AxisX.monitoring.superimposedBusy := FALSE;
   cmCathodeMainPnP1AxisX.monitoring.superimposedDone := FALSE;
   cmCathodeMainPnP1AxisX.monitoring.superimposedAborted := FALSE;
   cmCathodeMainPnP1AxisX.monitoring.selectSetPosition := 0;
   cmCathodeMainPnP1AxisX.monitoring.selectionController := FALSE;
   cmCathodeMainPnP1AxisX.monitoring.interlockGeneral := TRUE;
   cmCathodeMainPnP1AxisX.monitoring.interlockJogForward := TRUE;
   cmCathodeMainPnP1AxisX.monitoring.interlockJogBackward := TRUE;
   cmCathodeMainPnP1AxisX.monitoring.interlockWarningGeneral := FALSE;
   cmCathodeMainPnP1AxisX.monitoring.interlockWarningJogForward := FALSE;
   cmCathodeMainPnP1AxisX.monitoring.interlockWarningJogBackward := FALSE;
   cmCathodeMainPnP1AxisX.monitoring.valid := TRUE;
   cmCathodeMainPnP1AxisX.monitoring.busy := TRUE;
   cmCathodeMainPnP1AxisX.monitoring.error := FALSE;
   cmCathodeMainPnP1AxisX.monitoring.status := 16#7002;
   cmCathodeMainPnP1AxisX.monitoring.subfunctionStatus := 16#0000;
   cmCathodeMainPnP1AxisX.monitoring.actualPosition := 540.0;
   cmCathodeMainPnP1AxisX.monitoring.actualSpeed := 0.0;
   cmCathodeMainPnP1AxisX.monitoring.speedUnit := 1062;
   cmCathodeMainPnP1AxisX.monitoring.positionUnit := 1013;
   cmCathodeMainPnP1AxisX.monitoring.axisStatus1 := 16#0240_10A1;
   cmCathodeMainPnP1AxisX.monitoring.axisStatus2 := 16#0000_0000;
   cmCathodeMainPnP1AxisX.monitoring.axisType := 1;
   cmCathodeMainPnP1AxisX.monitoring.maxVelocity := 2500.0;
   cmCathodeMainPnP1AxisX.monitoring.actualCurrent := 0.0;
   cmCathodeMainPnP1AxisX.monitoring.actualTorque := 0.0;
   cmCathodeMainPnP1AxisX.monitoring.velocityOverrideEnabled := FALSE;
   cmCathodeMainPnP1AxisX.monitoring.sinaParaError := FALSE;
   cmCathodeMainPnP1AxisX.monitoring.sinaParaStatus := 16#0000_0000;
   cmCathodeMainPnP1AxisX.configuration.referenceDesignator := WSTRING#'CathodeMainPnP1AxisX';
   cmCathodeMainPnP1AxisX.configuration.disableAlarms := FALSE;
   cmCathodeMainPnP1AxisX.configuration.masterControlPopUp := TRUE;
   cmCathodeMainPnP1AxisX.configuration.setPositions[0].position := 0.0;
   cmCathodeMainPnP1AxisX.configuration.setPositions[1].position := 540.0;
   cmCathodeMainPnP1AxisX.configuration.setPositions[2].position := 544.0;
   cmCathodeMainPnP1AxisX.configuration.setPositions[3..15].position := 0.0;
   cmCathodeMainPnP1AxisX.configuration.setPositions[0..1].velocity := 500.0;
   cmCathodeMainPnP1AxisX.configuration.setPositions[2].velocity := 30.0;
   cmCathodeMainPnP1AxisX.configuration.setPositions[3..15].velocity := -1.0;
   cmCathodeMainPnP1AxisX.configuration.setPositions[0..1].acceleration := 5000.0;
   cmCathodeMainPnP1AxisX.configuration.setPositions[2].acceleration := 30.0;
   cmCathodeMainPnP1AxisX.configuration.setPositions[3..15].acceleration := -1.0;
   cmCathodeMainPnP1AxisX.configuration.setPositions[0..1].deceleration := 5000.0;
   cmCathodeMainPnP1AxisX.configuration.setPositions[2].deceleration := 30.0;
   cmCathodeMainPnP1AxisX.configuration.setPositions[3..15].deceleration := -1.0;
   cmCathodeMainPnP1AxisX.configuration.setPositions[0..15]."name" := '';
   cmCathodeMainPnP2AxisX.commandConfiguration.generalSettings.stopOnError := TRUE;
   cmCathodeMainPnP2AxisX.commandConfiguration.generalSettings.resetWithRestart := FALSE;
   cmCathodeMainPnP2AxisX.commandConfiguration.generalSettings.abortWaitingSyncCmd := TRUE;
   cmCathodeMainPnP2AxisX.commandConfiguration.power.startMode := 1;
   cmCathodeMainPnP2AxisX.commandConfiguration.power.stopMode := 0;
   cmCathodeMainPnP2AxisX.commandConfiguration.power.syncMotionSimulation := FALSE;
   cmCathodeMainPnP2AxisX.commandConfiguration.power.syncMotionSimulationExtendedMode := -1;
   cmCathodeMainPnP2AxisX.commandConfiguration.jog.velocity := 10.0;
   cmCathodeMainPnP2AxisX.commandConfiguration.jog.acceleration := 100.0;
   cmCathodeMainPnP2AxisX.commandConfiguration.jog.deceleration := 100.0;
   cmCathodeMainPnP2AxisX.commandConfiguration.jog.jerk := -1.0;
   cmCathodeMainPnP2AxisX.commandConfiguration.jog.positionControlled := TRUE;
   cmCathodeMainPnP2AxisX.commandConfiguration.jog.increment := 0.0;
   cmCathodeMainPnP2AxisX.commandConfiguration.jog.mode := 0;
   cmCathodeMainPnP2AxisX.commandConfiguration.moveVelocity.velocity := 10.0;
   cmCathodeMainPnP2AxisX.commandConfiguration.moveVelocity.acceleration := 100.0;
   cmCathodeMainPnP2AxisX.commandConfiguration.moveVelocity.deceleration := 100.0;
   cmCathodeMainPnP2AxisX.commandConfiguration.moveVelocity.jerk := -1.0;
   cmCathodeMainPnP2AxisX.commandConfiguration.moveVelocity.direction := 0;
   cmCathodeMainPnP2AxisX.commandConfiguration.moveVelocity.positionControlled := TRUE;
   cmCathodeMainPnP2AxisX.commandConfiguration.moveVelocity.velocityChangeOnTheFly := FALSE;
   cmCathodeMainPnP2AxisX.commandConfiguration.stop.deceleration := -1.0;
   cmCathodeMainPnP2AxisX.commandConfiguration.stop.jerk := -1.0;
   cmCathodeMainPnP2AxisX.commandConfiguration.stop.abortAcceleration := FALSE;
   cmCathodeMainPnP2AxisX.commandConfiguration.fastStop.deceleration := -1.0;
   cmCathodeMainPnP2AxisX.commandConfiguration.fastStop.jerk := -1.0;
   cmCathodeMainPnP2AxisX.commandConfiguration.fastStop.abortAcceleration := FALSE;
   cmCathodeMainPnP2AxisX.commandConfiguration.fastStop.replaceStopPossible := FALSE;
   cmCathodeMainPnP2AxisX.commandConfiguration.torqueLimiting.limit := -1.0;
   cmCathodeMainPnP2AxisX.commandConfiguration.torqueLimiting.mode := 0;
   cmCathodeMainPnP2AxisX.commandConfiguration.homing.position := 0.0;
   cmCathodeMainPnP2AxisX.commandConfiguration.homing.mode := 0;
   cmCathodeMainPnP2AxisX.commandConfiguration.homing.sensor := 0;
   cmCathodeMainPnP2AxisX.commandConfiguration.homing.extendedMode := -1;
   cmCathodeMainPnP2AxisX.commandConfiguration.homing.extendedModeTorqueLimit := 0.0;
   cmCathodeMainPnP2AxisX.commandConfiguration.homing.extendedModeTargetPosition := 0.0;
   cmCathodeMainPnP2AxisX.commandConfiguration.posRelative.distance := 0.0;
   cmCathodeMainPnP2AxisX.commandConfiguration.posRelative.velocity := 10.0;
   cmCathodeMainPnP2AxisX.commandConfiguration.posRelative.acceleration := 100.0;
   cmCathodeMainPnP2AxisX.commandConfiguration.posRelative.deceleration := 100.0;
   cmCathodeMainPnP2AxisX.commandConfiguration.posRelative.jerk := -1.0;
   cmCathodeMainPnP2AxisX.commandConfiguration.posRelative.direction := 0;
   cmCathodeMainPnP2AxisX.commandConfiguration.posAbsolute.position := 0.0;
   cmCathodeMainPnP2AxisX.commandConfiguration.posAbsolute.velocity := -1.0;
   cmCathodeMainPnP2AxisX.commandConfiguration.posAbsolute.acceleration := -1.0;
   cmCathodeMainPnP2AxisX.commandConfiguration.posAbsolute.deceleration := -1.0;
   cmCathodeMainPnP2AxisX.commandConfiguration.posAbsolute.jerk := 1382.07275733567;
   cmCathodeMainPnP2AxisX.commandConfiguration.posAbsolute.direction := 1;
   cmCathodeMainPnP2AxisX.commandConfiguration.posAbsolute.positionChangeOnTheFly := FALSE;
   cmCathodeMainPnP2AxisX.commandConfiguration.posAbsolute.velocityChangeOnTheFly := FALSE;
   cmCathodeMainPnP2AxisX.commandConfiguration.posSuperimposed.distance := 0.0;
   cmCathodeMainPnP2AxisX.commandConfiguration.posSuperimposed.velocityDiff := -1.0;
   cmCathodeMainPnP2AxisX.commandConfiguration.posSuperimposed.acceleration := -1.0;
   cmCathodeMainPnP2AxisX.commandConfiguration.posSuperimposed.deceleration := -1.0;
   cmCathodeMainPnP2AxisX.commandConfiguration.posSuperimposed.jerk := -1.0;
   cmCathodeMainPnP2AxisX.commandConfiguration.posSuperimposed.direction := 0;
   cmCathodeMainPnP2AxisX.commandConfiguration.haltSuperimposed.deceleration := -1.0;
   cmCathodeMainPnP2AxisX.commandConfiguration.haltSuperimposed.jerk := -1.0;
   cmCathodeMainPnP2AxisX.commandConfiguration.haltSuperimposed.abortAcceleration := FALSE;
   cmCathodeMainPnP2AxisX.commandConfiguration.gearInRelative.ratioNumerator := 1;
   cmCathodeMainPnP2AxisX.commandConfiguration.gearInRelative.ratioDenominator := 1;
   cmCathodeMainPnP2AxisX.commandConfiguration.gearInRelative.acceleration := -1.0;
   cmCathodeMainPnP2AxisX.commandConfiguration.gearInRelative.deceleration := -1.0;
   cmCathodeMainPnP2AxisX.commandConfiguration.gearInRelative.jerk := -1.0;
   cmCathodeMainPnP2AxisX.commandConfiguration.gearInRelative.ratioChangeOnTheFly := FALSE;
   cmCathodeMainPnP2AxisX.commandConfiguration.gearInAbsolute.ratioNumerator := 1;
   cmCathodeMainPnP2AxisX.commandConfiguration.gearInAbsolute.ratioDenominator := 1;
   cmCathodeMainPnP2AxisX.commandConfiguration.gearInAbsolute.masterSyncPosition := 0.0;
   cmCathodeMainPnP2AxisX.commandConfiguration.gearInAbsolute.slaveSyncPosition := 0.0;
   cmCathodeMainPnP2AxisX.commandConfiguration.gearInAbsolute.syncProfileReference := 1;
   cmCathodeMainPnP2AxisX.commandConfiguration.gearInAbsolute.masterStartDistance := 0.0;
   cmCathodeMainPnP2AxisX.commandConfiguration.gearInAbsolute.velocity := -1.0;
   cmCathodeMainPnP2AxisX.commandConfiguration.gearInAbsolute.acceleration := -1.0;
   cmCathodeMainPnP2AxisX.commandConfiguration.gearInAbsolute.deceleration := -1.0;
   cmCathodeMainPnP2AxisX.commandConfiguration.gearInAbsolute.jerk := -1.0;
   cmCathodeMainPnP2AxisX.commandConfiguration.gearInAbsolute.syncDirection := 1;
   cmCathodeMainPnP2AxisX.commandConfiguration.gearInAbsolute.ratioChangeOnTheFly := FALSE;
   cmCathodeMainPnP2AxisX.commandConfiguration.gearInVelocity.continuousUpdate := FALSE;
   cmCathodeMainPnP2AxisX.commandConfiguration.gearInVelocity.ratioNumerator := 1;
   cmCathodeMainPnP2AxisX.commandConfiguration.gearInVelocity.ratioDenominator := 1;
   cmCathodeMainPnP2AxisX.commandConfiguration.gearInVelocity.acceleration := -1.0;
   cmCathodeMainPnP2AxisX.commandConfiguration.gearInVelocity.deceleration := -1.0;
   cmCathodeMainPnP2AxisX.commandConfiguration.gearInVelocity.jerk := -1.0;
   cmCathodeMainPnP2AxisX.commandConfiguration.gearInVelocity.positionControlled := FALSE;
   cmCathodeMainPnP2AxisX.commandConfiguration.camIn.masterOffset := 0.0;
   cmCathodeMainPnP2AxisX.commandConfiguration.camIn.slaveOffset := 0.0;
   cmCathodeMainPnP2AxisX.commandConfiguration.camIn.masterScaling := 1.0;
   cmCathodeMainPnP2AxisX.commandConfiguration.camIn.slaveScaling := 1.0;
   cmCathodeMainPnP2AxisX.commandConfiguration.camIn.masterSyncPosition := 0.0;
   cmCathodeMainPnP2AxisX.commandConfiguration.camIn.syncProfileReference := 1;
   cmCathodeMainPnP2AxisX.commandConfiguration.camIn.masterStartDistance := 0.0;
   cmCathodeMainPnP2AxisX.commandConfiguration.camIn.velocity := -1.0;
   cmCathodeMainPnP2AxisX.commandConfiguration.camIn.acceleration := -1.0;
   cmCathodeMainPnP2AxisX.commandConfiguration.camIn.deceleration := -1.0;
   cmCathodeMainPnP2AxisX.commandConfiguration.camIn.jerk := -1.0;
   cmCathodeMainPnP2AxisX.commandConfiguration.camIn.applicationMode := 0;
   cmCathodeMainPnP2AxisX.commandConfiguration.camIn.syncDirection := 1;
   cmCathodeMainPnP2AxisX.commandConfiguration.gearOutCamOut.slavePosition := 0.0;
   cmCathodeMainPnP2AxisX.commandConfiguration.gearOutCamOut.syncProfileReference := 1;
   cmCathodeMainPnP2AxisX.commandConfiguration.gearOutCamOut.masterStopDistance := 0.0;
   cmCathodeMainPnP2AxisX.commandConfiguration.gearOutCamOut.deceleration := -1.0;
   cmCathodeMainPnP2AxisX.commandConfiguration.gearOutCamOut.jerk := -1.0;
   cmCathodeMainPnP2AxisX.commandConfiguration.gearOutCamOut.syncOutDirection := 3;
   cmCathodeMainPnP2AxisX.commandConfiguration.gearOutCamOut.gearOutCamOutMode := -1;
   cmCathodeMainPnP2AxisX.commandConfiguration.phasing.phaseShift := 0.0;
   cmCathodeMainPnP2AxisX.commandConfiguration.phasing.velocity := -1.0;
   cmCathodeMainPnP2AxisX.commandConfiguration.phasing.acceleration := -1.0;
   cmCathodeMainPnP2AxisX.commandConfiguration.phasing.deceleration := -1.0;
   cmCathodeMainPnP2AxisX.commandConfiguration.phasing.jerk := -1.0;
   cmCathodeMainPnP2AxisX.commandConfiguration.phasing.profileReference := 0;
   cmCathodeMainPnP2AxisX.commandConfiguration.phasing.phasingDistance := 0.0;
   cmCathodeMainPnP2AxisX.commandConfiguration.phasing.startPosition := 0.0;
   cmCathodeMainPnP2AxisX.commandConfiguration.phasing.direction := 3;
   cmCathodeMainPnP2AxisX.commandConfiguration.phasing.phaseAbsolute := TRUE;
   cmCathodeMainPnP2AxisX.commandConfiguration.phasing.phaseShiftChangeOnTheFly := FALSE;
   cmCathodeMainPnP2AxisX.commandConfiguration.offset.offset := 0.0;
   cmCathodeMainPnP2AxisX.commandConfiguration.offset.profileReference := 1;
   cmCathodeMainPnP2AxisX.commandConfiguration.offset.offsetDistance := 0.0;
   cmCathodeMainPnP2AxisX.commandConfiguration.offset.startPosition := 0.0;
   cmCathodeMainPnP2AxisX.commandConfiguration.offset.direction := 3;
   cmCathodeMainPnP2AxisX.commandConfiguration.offset.offsetAbsolute := TRUE;
   cmCathodeMainPnP2AxisX.commandConfiguration.offset.offsetChangeOnTheFly := FALSE;
   cmCathodeMainPnP2AxisX.commands.enableMasterControl := TRUE;
   cmCathodeMainPnP2AxisX.commands.enableAxis := FALSE;
   cmCathodeMainPnP2AxisX.commands.resetAxis := FALSE;
   cmCathodeMainPnP2AxisX.commands.openBrake := FALSE;
   cmCathodeMainPnP2AxisX.commands.jogForward := FALSE;
   cmCathodeMainPnP2AxisX.commands.jogBackward := FALSE;
   cmCathodeMainPnP2AxisX.commands.moveVelocity := FALSE;
   cmCathodeMainPnP2AxisX.commands.stop := FALSE;
   cmCathodeMainPnP2AxisX.commands.fastStop := FALSE;
   cmCathodeMainPnP2AxisX.commands.torqueLimiting := FALSE;
   cmCathodeMainPnP2AxisX.commands.homing := FALSE;
   cmCathodeMainPnP2AxisX.commands.posRelative := FALSE;
   cmCathodeMainPnP2AxisX.commands.posAbsolute := FALSE;
   cmCathodeMainPnP2AxisX.commands.posSuperimposed := FALSE;
   cmCathodeMainPnP2AxisX.commands.haltSuperimposed := FALSE;
   cmCathodeMainPnP2AxisX.commands.selectSetPosition := 0;
   cmCathodeMainPnP2AxisX.commands.uploadParameters := FALSE;
   cmCathodeMainPnP2AxisX.commands.refreshConfiguration := FALSE;
   cmCathodeMainPnP2AxisX.commands.editConfiguration := FALSE;
   cmCathodeMainPnP2AxisX.commands.saveConfiguration := FALSE;
   cmCathodeMainPnP2AxisX.commands.uploadCurrentTorque := FALSE;
   cmCathodeMainPnP2AxisX.commands.reset := FALSE;
   cmCathodeMainPnP2AxisX.monitoring.enable := TRUE;
   cmCathodeMainPnP2AxisX.monitoring.referenceDesignator := WSTRING#'CathodeMainPnP2AxisX';
   cmCathodeMainPnP2AxisX.monitoring.enabled := TRUE;
   cmCathodeMainPnP2AxisX.monitoring.enableManualCmds := FALSE;
   cmCathodeMainPnP2AxisX.monitoring.reset := FALSE;
   cmCathodeMainPnP2AxisX.monitoring.resetAxis := FALSE;
   cmCathodeMainPnP2AxisX.monitoring.enableAxis := TRUE;
   cmCathodeMainPnP2AxisX.monitoring.openBrake := FALSE;
   cmCathodeMainPnP2AxisX.monitoring.jogBackward := FALSE;
   cmCathodeMainPnP2AxisX.monitoring.jogForward := FALSE;
   cmCathodeMainPnP2AxisX.monitoring.moveVelocity := FALSE;
   cmCathodeMainPnP2AxisX.monitoring.stop := FALSE;
   cmCathodeMainPnP2AxisX.monitoring.fastStop := FALSE;
   cmCathodeMainPnP2AxisX.monitoring.torqueLimiting := FALSE;
   cmCathodeMainPnP2AxisX.monitoring.homing := FALSE;
   cmCathodeMainPnP2AxisX.monitoring.posRelative := FALSE;
   cmCathodeMainPnP2AxisX.monitoring.posAbsolute := FALSE;
   cmCathodeMainPnP2AxisX.monitoring.posSuperimposed := FALSE;
   cmCathodeMainPnP2AxisX.monitoring.haltSuperimposed := FALSE;
   cmCathodeMainPnP2AxisX.monitoring.brakeOpened := FALSE;
   cmCathodeMainPnP2AxisX.monitoring.axisEnabled := TRUE;
   cmCathodeMainPnP2AxisX.monitoring.resetActive := FALSE;
   cmCathodeMainPnP2AxisX.monitoring.inVelocity := FALSE;
   cmCathodeMainPnP2AxisX.monitoring.inLimitation := FALSE;
   cmCathodeMainPnP2AxisX.monitoring.inClamping := FALSE;
   cmCathodeMainPnP2AxisX.monitoring.startSync := FALSE;
   cmCathodeMainPnP2AxisX.monitoring.inSync := FALSE;
   cmCathodeMainPnP2AxisX.monitoring.inSimulation := FALSE;
   cmCathodeMainPnP2AxisX.monitoring.jogSelected := FALSE;
   cmCathodeMainPnP2AxisX.monitoring.moveVelocitySelected := FALSE;
   cmCathodeMainPnP2AxisX.monitoring.stopSelected := FALSE;
   cmCathodeMainPnP2AxisX.monitoring.fastStopSelected := FALSE;
   cmCathodeMainPnP2AxisX.monitoring.torqueLimitingSelected := FALSE;
   cmCathodeMainPnP2AxisX.monitoring.homingSelected := FALSE;
   cmCathodeMainPnP2AxisX.monitoring.posRelativeSelected := FALSE;
   cmCathodeMainPnP2AxisX.monitoring.posAbsoluteSelected := FALSE;
   cmCathodeMainPnP2AxisX.monitoring.posSuperimposedSelected := FALSE;
   cmCathodeMainPnP2AxisX.monitoring.haltSuperimposedSelected := FALSE;
   cmCathodeMainPnP2AxisX.monitoring.commandBusy := FALSE;
   cmCathodeMainPnP2AxisX.monitoring.commandDone := FALSE;
   cmCathodeMainPnP2AxisX.monitoring.commandAborted := FALSE;
   cmCathodeMainPnP2AxisX.monitoring.homingCommandBusy := FALSE;
   cmCathodeMainPnP2AxisX.monitoring.homingCommandDone := FALSE;
   cmCathodeMainPnP2AxisX.monitoring.homingCommandAborted := FALSE;
   cmCathodeMainPnP2AxisX.monitoring.superimposedBusy := FALSE;
   cmCathodeMainPnP2AxisX.monitoring.superimposedDone := FALSE;
   cmCathodeMainPnP2AxisX.monitoring.superimposedAborted := FALSE;
   cmCathodeMainPnP2AxisX.monitoring.selectSetPosition := 0;
   cmCathodeMainPnP2AxisX.monitoring.selectionController := FALSE;
   cmCathodeMainPnP2AxisX.monitoring.interlockGeneral := TRUE;
   cmCathodeMainPnP2AxisX.monitoring.interlockJogForward := TRUE;
   cmCathodeMainPnP2AxisX.monitoring.interlockJogBackward := TRUE;
   cmCathodeMainPnP2AxisX.monitoring.interlockWarningGeneral := FALSE;
   cmCathodeMainPnP2AxisX.monitoring.interlockWarningJogForward := FALSE;
   cmCathodeMainPnP2AxisX.monitoring.interlockWarningJogBackward := FALSE;
   cmCathodeMainPnP2AxisX.monitoring.valid := TRUE;
   cmCathodeMainPnP2AxisX.monitoring.busy := TRUE;
   cmCathodeMainPnP2AxisX.monitoring.error := FALSE;
   cmCathodeMainPnP2AxisX.monitoring.status := 16#7002;
   cmCathodeMainPnP2AxisX.monitoring.subfunctionStatus := 16#0000;
   cmCathodeMainPnP2AxisX.monitoring.actualPosition := 540.0;
   cmCathodeMainPnP2AxisX.monitoring.actualSpeed := 0.0;
   cmCathodeMainPnP2AxisX.monitoring.speedUnit := 1062;
   cmCathodeMainPnP2AxisX.monitoring.positionUnit := 1013;
   cmCathodeMainPnP2AxisX.monitoring.axisStatus1 := 16#0240_10A1;
   cmCathodeMainPnP2AxisX.monitoring.axisStatus2 := 16#0000_0000;
   cmCathodeMainPnP2AxisX.monitoring.axisType := 1;
   cmCathodeMainPnP2AxisX.monitoring.maxVelocity := 2500.0;
   cmCathodeMainPnP2AxisX.monitoring.actualCurrent := 0.0;
   cmCathodeMainPnP2AxisX.monitoring.actualTorque := 0.0;
   cmCathodeMainPnP2AxisX.monitoring.velocityOverrideEnabled := FALSE;
   cmCathodeMainPnP2AxisX.monitoring.sinaParaError := FALSE;
   cmCathodeMainPnP2AxisX.monitoring.sinaParaStatus := 16#0000_0000;
   cmCathodeMainPnP2AxisX.configuration.referenceDesignator := WSTRING#'CathodeMainPnP2AxisX';
   cmCathodeMainPnP2AxisX.configuration.disableAlarms := FALSE;
   cmCathodeMainPnP2AxisX.configuration.masterControlPopUp := TRUE;
   cmCathodeMainPnP2AxisX.configuration.setPositions[0].position := 0.0;
   cmCathodeMainPnP2AxisX.configuration.setPositions[1].position := 540.0;
   cmCathodeMainPnP2AxisX.configuration.setPositions[2].position := 538.0;
   cmCathodeMainPnP2AxisX.configuration.setPositions[3..15].position := 0.0;
   cmCathodeMainPnP2AxisX.configuration.setPositions[0..1].velocity := 500.0;
   cmCathodeMainPnP2AxisX.configuration.setPositions[2].velocity := 30.0;
   cmCathodeMainPnP2AxisX.configuration.setPositions[3..15].velocity := -1.0;
   cmCathodeMainPnP2AxisX.configuration.setPositions[0..1].acceleration := 5000.0;
   cmCathodeMainPnP2AxisX.configuration.setPositions[2].acceleration := 30.0;
   cmCathodeMainPnP2AxisX.configuration.setPositions[3..15].acceleration := -1.0;
   cmCathodeMainPnP2AxisX.configuration.setPositions[0..1].deceleration := 5000.0;
   cmCathodeMainPnP2AxisX.configuration.setPositions[2].deceleration := 30.0;
   cmCathodeMainPnP2AxisX.configuration.setPositions[3..15].deceleration := -1.0;
   cmCathodeMainPnP2AxisX.configuration.setPositions[0..15]."name" := '';
   cmCathodeMainPnP1AxisY.commandConfiguration.generalSettings.stopOnError := TRUE;
   cmCathodeMainPnP1AxisY.commandConfiguration.generalSettings.resetWithRestart := FALSE;
   cmCathodeMainPnP1AxisY.commandConfiguration.generalSettings.abortWaitingSyncCmd := TRUE;
   cmCathodeMainPnP1AxisY.commandConfiguration.power.startMode := 1;
   cmCathodeMainPnP1AxisY.commandConfiguration.power.stopMode := 0;
   cmCathodeMainPnP1AxisY.commandConfiguration.power.syncMotionSimulation := FALSE;
   cmCathodeMainPnP1AxisY.commandConfiguration.power.syncMotionSimulationExtendedMode := -1;
   cmCathodeMainPnP1AxisY.commandConfiguration.jog.velocity := 10.0;
   cmCathodeMainPnP1AxisY.commandConfiguration.jog.acceleration := 100.0;
   cmCathodeMainPnP1AxisY.commandConfiguration.jog.deceleration := 100.0;
   cmCathodeMainPnP1AxisY.commandConfiguration.jog.jerk := -1.0;
   cmCathodeMainPnP1AxisY.commandConfiguration.jog.positionControlled := TRUE;
   cmCathodeMainPnP1AxisY.commandConfiguration.jog.increment := 0.0;
   cmCathodeMainPnP1AxisY.commandConfiguration.jog.mode := 0;
   cmCathodeMainPnP1AxisY.commandConfiguration.moveVelocity.velocity := 10.0;
   cmCathodeMainPnP1AxisY.commandConfiguration.moveVelocity.acceleration := 100.0;
   cmCathodeMainPnP1AxisY.commandConfiguration.moveVelocity.deceleration := 100.0;
   cmCathodeMainPnP1AxisY.commandConfiguration.moveVelocity.jerk := 0.0;
   cmCathodeMainPnP1AxisY.commandConfiguration.moveVelocity.direction := 0;
   cmCathodeMainPnP1AxisY.commandConfiguration.moveVelocity.positionControlled := TRUE;
   cmCathodeMainPnP1AxisY.commandConfiguration.moveVelocity.velocityChangeOnTheFly := FALSE;
   cmCathodeMainPnP1AxisY.commandConfiguration.stop.deceleration := -1.0;
   cmCathodeMainPnP1AxisY.commandConfiguration.stop.jerk := -1.0;
   cmCathodeMainPnP1AxisY.commandConfiguration.stop.abortAcceleration := FALSE;
   cmCathodeMainPnP1AxisY.commandConfiguration.fastStop.deceleration := -1.0;
   cmCathodeMainPnP1AxisY.commandConfiguration.fastStop.jerk := -1.0;
   cmCathodeMainPnP1AxisY.commandConfiguration.fastStop.abortAcceleration := FALSE;
   cmCathodeMainPnP1AxisY.commandConfiguration.fastStop.replaceStopPossible := FALSE;
   cmCathodeMainPnP1AxisY.commandConfiguration.torqueLimiting.limit := -1.0;
   cmCathodeMainPnP1AxisY.commandConfiguration.torqueLimiting.mode := 0;
   cmCathodeMainPnP1AxisY.commandConfiguration.homing.position := 0.0;
   cmCathodeMainPnP1AxisY.commandConfiguration.homing.mode := 0;
   cmCathodeMainPnP1AxisY.commandConfiguration.homing.sensor := 0;
   cmCathodeMainPnP1AxisY.commandConfiguration.homing.extendedMode := -1;
   cmCathodeMainPnP1AxisY.commandConfiguration.homing.extendedModeTorqueLimit := 0.0;
   cmCathodeMainPnP1AxisY.commandConfiguration.homing.extendedModeTargetPosition := 0.0;
   cmCathodeMainPnP1AxisY.commandConfiguration.posRelative.distance := 0.0;
   cmCathodeMainPnP1AxisY.commandConfiguration.posRelative.velocity := 10.0;
   cmCathodeMainPnP1AxisY.commandConfiguration.posRelative.acceleration := 100.0;
   cmCathodeMainPnP1AxisY.commandConfiguration.posRelative.deceleration := 100.0;
   cmCathodeMainPnP1AxisY.commandConfiguration.posRelative.jerk := 0.0;
   cmCathodeMainPnP1AxisY.commandConfiguration.posRelative.direction := 0;
   cmCathodeMainPnP1AxisY.commandConfiguration.posAbsolute.position := 0.0;
   cmCathodeMainPnP1AxisY.commandConfiguration.posAbsolute.velocity := 0.0;
   cmCathodeMainPnP1AxisY.commandConfiguration.posAbsolute.acceleration := -1.0;
   cmCathodeMainPnP1AxisY.commandConfiguration.posAbsolute.deceleration := -1.0;
   cmCathodeMainPnP1AxisY.commandConfiguration.posAbsolute.jerk := 0.0;
   cmCathodeMainPnP1AxisY.commandConfiguration.posAbsolute.direction := 1;
   cmCathodeMainPnP1AxisY.commandConfiguration.posAbsolute.positionChangeOnTheFly := FALSE;
   cmCathodeMainPnP1AxisY.commandConfiguration.posAbsolute.velocityChangeOnTheFly := FALSE;
   cmCathodeMainPnP1AxisY.commandConfiguration.posSuperimposed.distance := 0.0;
   cmCathodeMainPnP1AxisY.commandConfiguration.posSuperimposed.velocityDiff := -1.0;
   cmCathodeMainPnP1AxisY.commandConfiguration.posSuperimposed.acceleration := -1.0;
   cmCathodeMainPnP1AxisY.commandConfiguration.posSuperimposed.deceleration := -1.0;
   cmCathodeMainPnP1AxisY.commandConfiguration.posSuperimposed.jerk := -1.0;
   cmCathodeMainPnP1AxisY.commandConfiguration.posSuperimposed.direction := 0;
   cmCathodeMainPnP1AxisY.commandConfiguration.haltSuperimposed.deceleration := -1.0;
   cmCathodeMainPnP1AxisY.commandConfiguration.haltSuperimposed.jerk := -1.0;
   cmCathodeMainPnP1AxisY.commandConfiguration.haltSuperimposed.abortAcceleration := FALSE;
   cmCathodeMainPnP1AxisY.commandConfiguration.gearInRelative.ratioNumerator := 1;
   cmCathodeMainPnP1AxisY.commandConfiguration.gearInRelative.ratioDenominator := 1;
   cmCathodeMainPnP1AxisY.commandConfiguration.gearInRelative.acceleration := -1.0;
   cmCathodeMainPnP1AxisY.commandConfiguration.gearInRelative.deceleration := -1.0;
   cmCathodeMainPnP1AxisY.commandConfiguration.gearInRelative.jerk := -1.0;
   cmCathodeMainPnP1AxisY.commandConfiguration.gearInRelative.ratioChangeOnTheFly := FALSE;
   cmCathodeMainPnP1AxisY.commandConfiguration.gearInAbsolute.ratioNumerator := 1;
   cmCathodeMainPnP1AxisY.commandConfiguration.gearInAbsolute.ratioDenominator := 1;
   cmCathodeMainPnP1AxisY.commandConfiguration.gearInAbsolute.masterSyncPosition := 0.0;
   cmCathodeMainPnP1AxisY.commandConfiguration.gearInAbsolute.slaveSyncPosition := 0.0;
   cmCathodeMainPnP1AxisY.commandConfiguration.gearInAbsolute.syncProfileReference := 1;
   cmCathodeMainPnP1AxisY.commandConfiguration.gearInAbsolute.masterStartDistance := 0.0;
   cmCathodeMainPnP1AxisY.commandConfiguration.gearInAbsolute.velocity := -1.0;
   cmCathodeMainPnP1AxisY.commandConfiguration.gearInAbsolute.acceleration := -1.0;
   cmCathodeMainPnP1AxisY.commandConfiguration.gearInAbsolute.deceleration := -1.0;
   cmCathodeMainPnP1AxisY.commandConfiguration.gearInAbsolute.jerk := -1.0;
   cmCathodeMainPnP1AxisY.commandConfiguration.gearInAbsolute.syncDirection := 1;
   cmCathodeMainPnP1AxisY.commandConfiguration.gearInAbsolute.ratioChangeOnTheFly := FALSE;
   cmCathodeMainPnP1AxisY.commandConfiguration.gearInVelocity.continuousUpdate := FALSE;
   cmCathodeMainPnP1AxisY.commandConfiguration.gearInVelocity.ratioNumerator := 1;
   cmCathodeMainPnP1AxisY.commandConfiguration.gearInVelocity.ratioDenominator := 1;
   cmCathodeMainPnP1AxisY.commandConfiguration.gearInVelocity.acceleration := -1.0;
   cmCathodeMainPnP1AxisY.commandConfiguration.gearInVelocity.deceleration := -1.0;
   cmCathodeMainPnP1AxisY.commandConfiguration.gearInVelocity.jerk := -1.0;
   cmCathodeMainPnP1AxisY.commandConfiguration.gearInVelocity.positionControlled := FALSE;
   cmCathodeMainPnP1AxisY.commandConfiguration.camIn.masterOffset := 0.0;
   cmCathodeMainPnP1AxisY.commandConfiguration.camIn.slaveOffset := 0.0;
   cmCathodeMainPnP1AxisY.commandConfiguration.camIn.masterScaling := 1.0;
   cmCathodeMainPnP1AxisY.commandConfiguration.camIn.slaveScaling := 1.0;
   cmCathodeMainPnP1AxisY.commandConfiguration.camIn.masterSyncPosition := 0.0;
   cmCathodeMainPnP1AxisY.commandConfiguration.camIn.syncProfileReference := 1;
   cmCathodeMainPnP1AxisY.commandConfiguration.camIn.masterStartDistance := 0.0;
   cmCathodeMainPnP1AxisY.commandConfiguration.camIn.velocity := -1.0;
   cmCathodeMainPnP1AxisY.commandConfiguration.camIn.acceleration := -1.0;
   cmCathodeMainPnP1AxisY.commandConfiguration.camIn.deceleration := -1.0;
   cmCathodeMainPnP1AxisY.commandConfiguration.camIn.jerk := -1.0;
   cmCathodeMainPnP1AxisY.commandConfiguration.camIn.applicationMode := 0;
   cmCathodeMainPnP1AxisY.commandConfiguration.camIn.syncDirection := 1;
   cmCathodeMainPnP1AxisY.commandConfiguration.gearOutCamOut.slavePosition := 0.0;
   cmCathodeMainPnP1AxisY.commandConfiguration.gearOutCamOut.syncProfileReference := 1;
   cmCathodeMainPnP1AxisY.commandConfiguration.gearOutCamOut.masterStopDistance := 0.0;
   cmCathodeMainPnP1AxisY.commandConfiguration.gearOutCamOut.deceleration := -1.0;
   cmCathodeMainPnP1AxisY.commandConfiguration.gearOutCamOut.jerk := -1.0;
   cmCathodeMainPnP1AxisY.commandConfiguration.gearOutCamOut.syncOutDirection := 3;
   cmCathodeMainPnP1AxisY.commandConfiguration.gearOutCamOut.gearOutCamOutMode := -1;
   cmCathodeMainPnP1AxisY.commandConfiguration.phasing.phaseShift := 0.0;
   cmCathodeMainPnP1AxisY.commandConfiguration.phasing.velocity := -1.0;
   cmCathodeMainPnP1AxisY.commandConfiguration.phasing.acceleration := -1.0;
   cmCathodeMainPnP1AxisY.commandConfiguration.phasing.deceleration := -1.0;
   cmCathodeMainPnP1AxisY.commandConfiguration.phasing.jerk := -1.0;
   cmCathodeMainPnP1AxisY.commandConfiguration.phasing.profileReference := 0;
   cmCathodeMainPnP1AxisY.commandConfiguration.phasing.phasingDistance := 0.0;
   cmCathodeMainPnP1AxisY.commandConfiguration.phasing.startPosition := 0.0;
   cmCathodeMainPnP1AxisY.commandConfiguration.phasing.direction := 3;
   cmCathodeMainPnP1AxisY.commandConfiguration.phasing.phaseAbsolute := TRUE;
   cmCathodeMainPnP1AxisY.commandConfiguration.phasing.phaseShiftChangeOnTheFly := FALSE;
   cmCathodeMainPnP1AxisY.commandConfiguration.offset.offset := 0.0;
   cmCathodeMainPnP1AxisY.commandConfiguration.offset.profileReference := 1;
   cmCathodeMainPnP1AxisY.commandConfiguration.offset.offsetDistance := 0.0;
   cmCathodeMainPnP1AxisY.commandConfiguration.offset.startPosition := 0.0;
   cmCathodeMainPnP1AxisY.commandConfiguration.offset.direction := 3;
   cmCathodeMainPnP1AxisY.commandConfiguration.offset.offsetAbsolute := TRUE;
   cmCathodeMainPnP1AxisY.commandConfiguration.offset.offsetChangeOnTheFly := FALSE;
   cmCathodeMainPnP1AxisY.commands.enableMasterControl := TRUE;
   cmCathodeMainPnP1AxisY.commands.enableAxis := FALSE;
   cmCathodeMainPnP1AxisY.commands.resetAxis := FALSE;
   cmCathodeMainPnP1AxisY.commands.openBrake := FALSE;
   cmCathodeMainPnP1AxisY.commands.jogForward := FALSE;
   cmCathodeMainPnP1AxisY.commands.jogBackward := FALSE;
   cmCathodeMainPnP1AxisY.commands.moveVelocity := FALSE;
   cmCathodeMainPnP1AxisY.commands.stop := FALSE;
   cmCathodeMainPnP1AxisY.commands.fastStop := FALSE;
   cmCathodeMainPnP1AxisY.commands.torqueLimiting := FALSE;
   cmCathodeMainPnP1AxisY.commands.homing := FALSE;
   cmCathodeMainPnP1AxisY.commands.posRelative := FALSE;
   cmCathodeMainPnP1AxisY.commands.posAbsolute := FALSE;
   cmCathodeMainPnP1AxisY.commands.posSuperimposed := FALSE;
   cmCathodeMainPnP1AxisY.commands.haltSuperimposed := FALSE;
   cmCathodeMainPnP1AxisY.commands.selectSetPosition := -1;
   cmCathodeMainPnP1AxisY.commands.uploadParameters := FALSE;
   cmCathodeMainPnP1AxisY.commands.refreshConfiguration := FALSE;
   cmCathodeMainPnP1AxisY.commands.editConfiguration := FALSE;
   cmCathodeMainPnP1AxisY.commands.saveConfiguration := FALSE;
   cmCathodeMainPnP1AxisY.commands.uploadCurrentTorque := FALSE;
   cmCathodeMainPnP1AxisY.commands.reset := FALSE;
   cmCathodeMainPnP1AxisY.monitoring.enable := TRUE;
   cmCathodeMainPnP1AxisY.monitoring.referenceDesignator := WSTRING#'CathodeMainPnP1AxisY';
   cmCathodeMainPnP1AxisY.monitoring.enabled := TRUE;
   cmCathodeMainPnP1AxisY.monitoring.enableManualCmds := FALSE;
   cmCathodeMainPnP1AxisY.monitoring.reset := FALSE;
   cmCathodeMainPnP1AxisY.monitoring.resetAxis := FALSE;
   cmCathodeMainPnP1AxisY.monitoring.enableAxis := TRUE;
   cmCathodeMainPnP1AxisY.monitoring.openBrake := FALSE;
   cmCathodeMainPnP1AxisY.monitoring.jogBackward := FALSE;
   cmCathodeMainPnP1AxisY.monitoring.jogForward := FALSE;
   cmCathodeMainPnP1AxisY.monitoring.moveVelocity := FALSE;
   cmCathodeMainPnP1AxisY.monitoring.stop := FALSE;
   cmCathodeMainPnP1AxisY.monitoring.fastStop := FALSE;
   cmCathodeMainPnP1AxisY.monitoring.torqueLimiting := FALSE;
   cmCathodeMainPnP1AxisY.monitoring.homing := FALSE;
   cmCathodeMainPnP1AxisY.monitoring.posRelative := FALSE;
   cmCathodeMainPnP1AxisY.monitoring.posAbsolute := FALSE;
   cmCathodeMainPnP1AxisY.monitoring.posSuperimposed := FALSE;
   cmCathodeMainPnP1AxisY.monitoring.haltSuperimposed := FALSE;
   cmCathodeMainPnP1AxisY.monitoring.brakeOpened := FALSE;
   cmCathodeMainPnP1AxisY.monitoring.axisEnabled := TRUE;
   cmCathodeMainPnP1AxisY.monitoring.resetActive := FALSE;
   cmCathodeMainPnP1AxisY.monitoring.inVelocity := FALSE;
   cmCathodeMainPnP1AxisY.monitoring.inLimitation := FALSE;
   cmCathodeMainPnP1AxisY.monitoring.inClamping := FALSE;
   cmCathodeMainPnP1AxisY.monitoring.startSync := FALSE;
   cmCathodeMainPnP1AxisY.monitoring.inSync := FALSE;
   cmCathodeMainPnP1AxisY.monitoring.inSimulation := FALSE;
   cmCathodeMainPnP1AxisY.monitoring.jogSelected := FALSE;
   cmCathodeMainPnP1AxisY.monitoring.moveVelocitySelected := FALSE;
   cmCathodeMainPnP1AxisY.monitoring.stopSelected := FALSE;
   cmCathodeMainPnP1AxisY.monitoring.fastStopSelected := FALSE;
   cmCathodeMainPnP1AxisY.monitoring.torqueLimitingSelected := FALSE;
   cmCathodeMainPnP1AxisY.monitoring.homingSelected := FALSE;
   cmCathodeMainPnP1AxisY.monitoring.posRelativeSelected := FALSE;
   cmCathodeMainPnP1AxisY.monitoring.posAbsoluteSelected := FALSE;
   cmCathodeMainPnP1AxisY.monitoring.posSuperimposedSelected := FALSE;
   cmCathodeMainPnP1AxisY.monitoring.haltSuperimposedSelected := FALSE;
   cmCathodeMainPnP1AxisY.monitoring.commandBusy := FALSE;
   cmCathodeMainPnP1AxisY.monitoring.commandDone := FALSE;
   cmCathodeMainPnP1AxisY.monitoring.commandAborted := FALSE;
   cmCathodeMainPnP1AxisY.monitoring.homingCommandBusy := FALSE;
   cmCathodeMainPnP1AxisY.monitoring.homingCommandDone := FALSE;
   cmCathodeMainPnP1AxisY.monitoring.homingCommandAborted := FALSE;
   cmCathodeMainPnP1AxisY.monitoring.superimposedBusy := FALSE;
   cmCathodeMainPnP1AxisY.monitoring.superimposedDone := FALSE;
   cmCathodeMainPnP1AxisY.monitoring.superimposedAborted := FALSE;
   cmCathodeMainPnP1AxisY.monitoring.selectSetPosition := -1;
   cmCathodeMainPnP1AxisY.monitoring.selectionController := FALSE;
   cmCathodeMainPnP1AxisY.monitoring.interlockGeneral := TRUE;
   cmCathodeMainPnP1AxisY.monitoring.interlockJogForward := TRUE;
   cmCathodeMainPnP1AxisY.monitoring.interlockJogBackward := TRUE;
   cmCathodeMainPnP1AxisY.monitoring.interlockWarningGeneral := FALSE;
   cmCathodeMainPnP1AxisY.monitoring.interlockWarningJogForward := FALSE;
   cmCathodeMainPnP1AxisY.monitoring.interlockWarningJogBackward := FALSE;
   cmCathodeMainPnP1AxisY.monitoring.valid := TRUE;
   cmCathodeMainPnP1AxisY.monitoring.busy := TRUE;
   cmCathodeMainPnP1AxisY.monitoring.error := FALSE;
   cmCathodeMainPnP1AxisY.monitoring.status := 16#7002;
   cmCathodeMainPnP1AxisY.monitoring.subfunctionStatus := 16#0000;
   cmCathodeMainPnP1AxisY.monitoring.actualPosition := 0.0;
   cmCathodeMainPnP1AxisY.monitoring.actualSpeed := 0.0;
   cmCathodeMainPnP1AxisY.monitoring.speedUnit := 1062;
   cmCathodeMainPnP1AxisY.monitoring.positionUnit := 1013;
   cmCathodeMainPnP1AxisY.monitoring.axisStatus1 := 16#0200_10E1;
   cmCathodeMainPnP1AxisY.monitoring.axisStatus2 := 16#0000_0000;
   cmCathodeMainPnP1AxisY.monitoring.axisType := 1;
   cmCathodeMainPnP1AxisY.monitoring.maxVelocity := 2500.0;
   cmCathodeMainPnP1AxisY.monitoring.actualCurrent := 0.0;
   cmCathodeMainPnP1AxisY.monitoring.actualTorque := 0.0;
   cmCathodeMainPnP1AxisY.monitoring.velocityOverrideEnabled := FALSE;
   cmCathodeMainPnP1AxisY.monitoring.sinaParaError := FALSE;
   cmCathodeMainPnP1AxisY.monitoring.sinaParaStatus := 16#0000_0000;
   cmCathodeMainPnP1AxisY.configuration.referenceDesignator := WSTRING#'CathodeMainPnP1AxisY';
   cmCathodeMainPnP1AxisY.configuration.disableAlarms := FALSE;
   cmCathodeMainPnP1AxisY.configuration.masterControlPopUp := TRUE;
   cmCathodeMainPnP1AxisY.configuration.setPositions[0..15].position := 0.0;
   cmCathodeMainPnP1AxisY.configuration.setPositions[0].velocity := 50.0;
   cmCathodeMainPnP1AxisY.configuration.setPositions[1].velocity := 30.0;
   cmCathodeMainPnP1AxisY.configuration.setPositions[2..15].velocity := -1.0;
   cmCathodeMainPnP1AxisY.configuration.setPositions[0].acceleration := 500.0;
   cmCathodeMainPnP1AxisY.configuration.setPositions[1].acceleration := 30.0;
   cmCathodeMainPnP1AxisY.configuration.setPositions[2..15].acceleration := -1.0;
   cmCathodeMainPnP1AxisY.configuration.setPositions[0].deceleration := 500.0;
   cmCathodeMainPnP1AxisY.configuration.setPositions[1].deceleration := 30.0;
   cmCathodeMainPnP1AxisY.configuration.setPositions[2..15].deceleration := -1.0;
   cmCathodeMainPnP1AxisY.configuration.setPositions[0..15]."name" := '';
   cmCathodeMainPnP1AxisZ.commandConfiguration.generalSettings.stopOnError := TRUE;
   cmCathodeMainPnP1AxisZ.commandConfiguration.generalSettings.resetWithRestart := FALSE;
   cmCathodeMainPnP1AxisZ.commandConfiguration.generalSettings.abortWaitingSyncCmd := TRUE;
   cmCathodeMainPnP1AxisZ.commandConfiguration.power.startMode := 1;
   cmCathodeMainPnP1AxisZ.commandConfiguration.power.stopMode := 0;
   cmCathodeMainPnP1AxisZ.commandConfiguration.power.syncMotionSimulation := FALSE;
   cmCathodeMainPnP1AxisZ.commandConfiguration.power.syncMotionSimulationExtendedMode := -1;
   cmCathodeMainPnP1AxisZ.commandConfiguration.jog.velocity := 10.0;
   cmCathodeMainPnP1AxisZ.commandConfiguration.jog.acceleration := 100.0;
   cmCathodeMainPnP1AxisZ.commandConfiguration.jog.deceleration := 100.0;
   cmCathodeMainPnP1AxisZ.commandConfiguration.jog.jerk := -1.0;
   cmCathodeMainPnP1AxisZ.commandConfiguration.jog.positionControlled := TRUE;
   cmCathodeMainPnP1AxisZ.commandConfiguration.jog.increment := 0.0;
   cmCathodeMainPnP1AxisZ.commandConfiguration.jog.mode := 0;
   cmCathodeMainPnP1AxisZ.commandConfiguration.moveVelocity.velocity := 10.0;
   cmCathodeMainPnP1AxisZ.commandConfiguration.moveVelocity.acceleration := 100.0;
   cmCathodeMainPnP1AxisZ.commandConfiguration.moveVelocity.deceleration := 100.0;
   cmCathodeMainPnP1AxisZ.commandConfiguration.moveVelocity.jerk := -1.0;
   cmCathodeMainPnP1AxisZ.commandConfiguration.moveVelocity.direction := 0;
   cmCathodeMainPnP1AxisZ.commandConfiguration.moveVelocity.positionControlled := TRUE;
   cmCathodeMainPnP1AxisZ.commandConfiguration.moveVelocity.velocityChangeOnTheFly := FALSE;
   cmCathodeMainPnP1AxisZ.commandConfiguration.stop.deceleration := -1.0;
   cmCathodeMainPnP1AxisZ.commandConfiguration.stop.jerk := -1.0;
   cmCathodeMainPnP1AxisZ.commandConfiguration.stop.abortAcceleration := FALSE;
   cmCathodeMainPnP1AxisZ.commandConfiguration.fastStop.deceleration := -1.0;
   cmCathodeMainPnP1AxisZ.commandConfiguration.fastStop.jerk := -1.0;
   cmCathodeMainPnP1AxisZ.commandConfiguration.fastStop.abortAcceleration := FALSE;
   cmCathodeMainPnP1AxisZ.commandConfiguration.fastStop.replaceStopPossible := FALSE;
   cmCathodeMainPnP1AxisZ.commandConfiguration.torqueLimiting.limit := -1.0;
   cmCathodeMainPnP1AxisZ.commandConfiguration.torqueLimiting.mode := 0;
   cmCathodeMainPnP1AxisZ.commandConfiguration.homing.position := 0.0;
   cmCathodeMainPnP1AxisZ.commandConfiguration.homing.mode := 0;
   cmCathodeMainPnP1AxisZ.commandConfiguration.homing.sensor := 0;
   cmCathodeMainPnP1AxisZ.commandConfiguration.homing.extendedMode := -1;
   cmCathodeMainPnP1AxisZ.commandConfiguration.homing.extendedModeTorqueLimit := 0.0;
   cmCathodeMainPnP1AxisZ.commandConfiguration.homing.extendedModeTargetPosition := 0.0;
   cmCathodeMainPnP1AxisZ.commandConfiguration.posRelative.distance := 0.0;
   cmCathodeMainPnP1AxisZ.commandConfiguration.posRelative.velocity := 10.0;
   cmCathodeMainPnP1AxisZ.commandConfiguration.posRelative.acceleration := 100.0;
   cmCathodeMainPnP1AxisZ.commandConfiguration.posRelative.deceleration := 100.0;
   cmCathodeMainPnP1AxisZ.commandConfiguration.posRelative.jerk := -1.0;
   cmCathodeMainPnP1AxisZ.commandConfiguration.posRelative.direction := 0;
   cmCathodeMainPnP1AxisZ.commandConfiguration.posAbsolute.position := 0.0;
   cmCathodeMainPnP1AxisZ.commandConfiguration.posAbsolute.velocity := -1.0;
   cmCathodeMainPnP1AxisZ.commandConfiguration.posAbsolute.acceleration := -1.0;
   cmCathodeMainPnP1AxisZ.commandConfiguration.posAbsolute.deceleration := -1.0;
   cmCathodeMainPnP1AxisZ.commandConfiguration.posAbsolute.jerk := -1.0;
   cmCathodeMainPnP1AxisZ.commandConfiguration.posAbsolute.direction := 1;
   cmCathodeMainPnP1AxisZ.commandConfiguration.posAbsolute.positionChangeOnTheFly := FALSE;
   cmCathodeMainPnP1AxisZ.commandConfiguration.posAbsolute.velocityChangeOnTheFly := FALSE;
   cmCathodeMainPnP1AxisZ.commandConfiguration.posSuperimposed.distance := 0.0;
   cmCathodeMainPnP1AxisZ.commandConfiguration.posSuperimposed.velocityDiff := -1.0;
   cmCathodeMainPnP1AxisZ.commandConfiguration.posSuperimposed.acceleration := -1.0;
   cmCathodeMainPnP1AxisZ.commandConfiguration.posSuperimposed.deceleration := -1.0;
